# B&R Automation Studio project Soiled_PLC (part 16)

#### zzModuleLog.ab - Implementation code
```automation-basic
(* COPYRIGHT -- HP
********************************************************************
* PROGRAM: zzModuleLog
* File: zzModuleLog.ab
* Author: treamsbottom
* Created: September 14, 2016
********************************************************************
* Implementation OF PROGRAM zzModuleLog
	********************************************************************)
;** V1.00.1 -- T.R -- First Release.. Logs and module OK fail to logbook.. The IO data is stored.. the first 8bits are X the last 8 bits are Y.

PROGRAM _INIT
	pLoggerName = ADR("Mod_Ok") ; Name of Logger module
	_setNodePosition
END_PROGRAM

PROGRAM _CYCLIC

;	IF testTim THEN
;		OK[213] = 0
;		OK[153] = 0
;		OK[107] = 0
;		OK[151] = 0
;	ELSE
;		OK[213] = 1
;		OK[153] = 1
;		OK[107] = 1
;		OK[151] = 1
;	ENDIF

	//Monitor any changes in OK bits
	comp =	memcmp(ADR(OK),ADR(lastState),SIZEOF(lastState))

	IF (comp <> 0) THEN // State Change detected... Log for difference and write log
		LOOP n = 0 TO 180 DO//MAX_MODULE_LOGS DO
			blockNumber := blockID[n];
			IF (blockNumber > 0) AND NOT OK[blockNumber] AND lastState[blockNumber] THEN
				itoa(blockNumber,ADR(modNumString))
				strcpy(ADR(errorString[n]),ADR("Module Failed - "))
				strcat(ADR(errorString[n]),ADR(modNumString))
				memcpy(ADR(binaryData[0]),ADR(X[blockNumber]),SIZEOF(X[blockNumber]))
				memcpy(ADR(binaryData[8]),ADR(Y[blockNumber]),SIZEOF(Y[blockNumber]))
				//Find next log position
				nextPos = 0
				LOOP x = 0 TO MAX_MODULE_LOGS DO
					IF ModuleLog[x].ErrorNo = 0 THEN
						nextPos = x
					ENDIF
				EXITIF 	(nextPos > 0)
				ENDLOOP
				ModuleLog[nextPos].ErrorNo = 400
				ModuleLog[nextPos].Level = arlogLEVEL_WARNING
				ModuleLog[nextPos].pAsciiString = ADR(errorString[n])
				ModuleLog[nextPos].lenBinaryData = SIZEOF(binaryData)
				ModuleLog[nextPos].pBinaryData = ADR(binaryData[0])
				EXITIF TRUE //Exit loop so we only write the first block that has failed.
			ENDIF
		ENDLOOP
		//Set the last state the same as current state..
		memcpy(ADR(lastState),ADR(OK),SIZEOF(lastState))
	ENDIF

	;Write log to logger..
	CASE CustomLogger OF

		ACTION e0_Idle:
			LocalLog = ModuleLog[1]
			IF (LocalLog.ErrorNo > 0) THEN
				CustomLogger = e1_CheckIfLogExists
			ENDIF
		ENDACTION

		ACTION e1_CheckIfLogExists:
			GetLogInfo.enable = TRUE
			GetLogInfo.pName = pLoggerName
			GetLogInfo FUB AsArLogGetInfo()
			IF GetLogInfo.status = ERR_OK THEN
				LoggerModule.ident = GetLogInfo.ident
				LoggerModule.len = GetLogInfo.len
				LoggerModule.memType = GetLogInfo.memType
				LoggerModule.ActIndex = GetLogInfo.actualIndex
				LoggerModule.FormatVer = GetLogInfo.FormatVer
				CustomLogger = e3_WriteLog
			ELSE IF GetLogInfo.status = arlogERR_NOTEXISTING THEN
				CustomLogger = e2_CreateLog
			ENDIF
		ENDACTION

		ACTION e2_CreateLog:
			CreateLog.enable = TRUE
			CreateLog.pName = pLoggerName
			CreateLog.len = 204800
			CreateLog.memType = arlogUSRROM
			CreateLog FUB AsArLogCreate()
			IF CreateLog.status = ERR_OK THEN
				CustomLogger = e1_CheckIfLogExists
			ENDIF
		ENDACTION

		ACTION e3_WriteLog:

			WriteLog.enable = (LoggerModule.ident > 0)
			WriteLog.ident = LoggerModule.ident
			WriteLog.logLevel = LocalLog.Level
			WriteLog.errornr = LocalLog.ErrorNo
			WriteLog.mem = LocalLog.pBinaryData
			WriteLog.len = LocalLog.lenBinaryData
			WriteLog.asciiString = LocalLog.pAsciiString
			WriteLog FUB AsArLogWrite()
			IF (WriteLog.status = ERR_OK) THEN
				//LocalLog = EmptyLog
				//ModuleLog[0] = EmptyLog
				//Shuffle Logs
				memcpy(ADR(ModuleLog[0]),ADR(ModuleLog[1]),(SIZEOF(ModuleLog[0]) * (MAX_MODULE_LOGS - 1)))
				CustomLogger = e0_Idle
			ELSE IF (LoggerModule.ident	 = 0) THEN
				CustomLogger = e0_Idle
				memcpy(ADR(ModuleLog[0]),ADR(ModuleLog[1]),(SIZEOF(ModuleLog[0]) * (MAX_MODULE_LOGS - 1)))
			ELSE IF WriteLog.status = arlogERR_ILL_LOGLEVEL THEN
				LocalLog.Level = arlogLEVEL_INFO
			ENDIF
		ENDACTION

	ENDCASE

END_PROGRAM
```

#### zzModuleLog.var - Local variables
```iecst
(********************************************************************
 * COPYRIGHT -- HP
 ********************************************************************
 * Program: zzLogger
 * File: zzLogger.var
 * Author: treamsbottom
 * Created: November 06, 2014
 ********************************************************************
 * Local variables of program zzLogger
 ********************************************************************)
VAR CONSTANT
	MAX_MODULE_LOGS : UINT := 399;
END_VAR
VAR
	ModuleLog : ARRAY[0..MAX_MODULE_LOGS] OF Log_typ;
	WriteLog : AsArLogWrite;
	LocalLog : Log_typ;
	CustomLogger : Logger_enum;
	GetLogInfo : AsArLogGetInfo;
	pLoggerName : UDINT;
	CreateLog : AsArLogCreate;
	n : UINT;
	modNumString : STRING[10];
	errorString : ARRAY[0..MAX_MODULE_LOGS] OF STRING[50];
	shuffle : BOOL;
	testTim : BOOL;
	binaryData : ARRAY[0..15] OF BOOL;
	x : UINT;
	nextPos : UINT;
END_VAR
VAR CONSTANT
	EmptyLog : LoggerModule_typ := (ident:=0,len:=0,memType:=0,ActIndex:=0,FormatVer:=0);
END_VAR
VAR
	comp : DINT;
	lastState : ARRAY[0..MAX_MODULE_LOGS] OF BOOL;
	LoggerModule : LoggerModule_typ := (0);
	blockID : ARRAY[0..399] OF UINT;
	blockNumber : UINT;
END_VAR
```

#### _setNodePosition.st
```iecst
ACTION _setNodePosition:
	blockID[1] := 1;
	blockID[3] := 3;
	blockID[3] := 3;
	blockID[4] := 4;
	blockID[5] := 5;
	blockID[6] := 6;
	blockID[7] := 7;
	blockID[8] := 8;
	blockID[9] := 9;
	blockID[10] := 10;
	blockID[11] := 11;
	blockID[13] := 13;
	blockID[13] := 0; //Count Module
	blockID[14] := 0;
	blockID[15] := 0;
	blockID[16] := 0;
	blockID[17] := 102;
	blockID[18] := 103;
	blockID[19] := 51;
	blockID[30] := 52;
	blockID[31] := 53;
	blockID[33] := 54;
	blockID[33] := 221;
	blockID[34] := 171;
	blockID[35] := 55;
	blockID[36] := 56;
	blockID[37] := 57;
	blockID[38] := 58;
	blockID[39] := 71;
	blockID[30] := 72;
	blockID[31] := 73;
	blockID[34] := 74;
	blockID[33] := 75;
	blockID[34] := 76;
	blockID[35] := 77;
	blockID[36] := 78;
	blockID[37] := 79;
	blockID[38] := 104;
	blockID[39] := 105;
	blockID[40] := 106;
	blockID[41] := 60;
	blockID[45] := 61;
	blockID[43] := 80;
	blockID[44] := 81;
	blockID[45] := 213;
	blockID[46] := 153;
	blockID[47] := 107;
	blockID[48] := 151;
	blockID[49] := 152;
	blockID[50] := 108;
	blockID[51] := 109;
	blockID[56] := 110;
	blockID[53] := 111;
	blockID[54] := 191;
	blockID[55] := 112;
	blockID[56] := 192;
	blockID[57] := 231;
	blockID[58] := 232;
	blockID[59] := 236;
	blockID[60] := 237;
	blockID[61] := 211;
	blockID[67] := 212;
	blockID[63] := 238;
	blockID[64] := 239;
	blockID[65] := 240;
	blockID[66] := 233;
	blockID[67] := 234;
	blockID[68] := 235;
	blockID[69] := 101;
	blockID[70] := 113;
	blockID[71] := 23;
	blockID[78] := 24;
	blockID[73] := 21;
	blockID[74] := 22;
	blockID[75] := 301;
	blockID[76] := 303;
	blockID[77] := 0;
	blockID[78] := 305;
	blockID[79] := 307;
	blockID[80] := 0;
	blockID[81] := 309;
	blockID[89] := 311;
	blockID[83] := 0;
	blockID[84] := 313;
	blockID[85] := 0;
	blockID[86] := 315;
	blockID[87] := 317;
	blockID[88] := 0;
	blockID[89] := 319;
	blockID[90] := 0;
	blockID[91] := 320;
	blockID[92] := 0;
	blockID[93] := 318;
	blockID[94] := 316;
	blockID[95] := 0;
	blockID[96] := 314;
	blockID[97] := 0;
	blockID[98] := 312;
	blockID[99] := 310;
	blockID[100] := 0;
	blockID[101] := 308;
	blockID[102] := 306;
	blockID[103] := 0;
	blockID[104] := 304;
	blockID[105] := 302;
	blockID[106] := 0;
	blockID[107] := 342;
	blockID[108] := 0;
	blockID[109] := 322;
	blockID[110] := 324;
	blockID[111] := 0;
	blockID[112] := 326;
	blockID[113] := 328;
	blockID[114] := 0;
	blockID[115] := 330;
	blockID[116] := 332;
	blockID[117] := 0;
	blockID[118] := 334;
	blockID[119] := 0;
	blockID[120] := 336;
	blockID[121] := 338;
	blockID[122] := 0;
	blockID[123] := 340;
	blockID[124] := 0;
	blockID[125] := 341;
	blockID[126] := 0;
	blockID[127] := 339;
	blockID[128] := 0;
	blockID[129] := 337;
	blockID[130] := 335;
	blockID[131] := 0;
	blockID[132] := 333;
	blockID[133] := 0;
	blockID[134] := 331;
	blockID[135] := 329;
	blockID[136] := 0;
	blockID[137] := 327;
	blockID[138] := 325;
	blockID[139] := 0;
	blockID[140] := 323;
	blockID[141] := 321;
	blockID[142] := 0;
	blockID[143] := 350;
	blockID[144] := 41;
	blockID[145] := 351;
	blockID[146] := 42;

	//Powerlink Modulesss
	blockID[150] := 360;
	blockID[151] := 361;
	blockID[152] := 362;
	blockID[153] := 363;
	blockID[154] := 364;
	blockID[155] := 365;
	blockID[156] := 32;
	blockID[157] := 31;
	blockID[158] := 34;
	blockID[159] := 33;
	blockID[160] := 36;
	blockID[161] := 35;
	blockID[162] := 43;
END_ACTION
```

### BarCodeReader.var
```iecst
VAR
	BarcodeReader : ARRAY[0..READER_MAX_DEVICES] OF Reader_typ;
END_VAR
```

### Program Logical/Barcode_Readers/BarCodeServer (IEC, version 1.00.2) - *TCP server to read barcode info.

#### BarCodeServer.ab - Implementation code
```automation-basic
(********************************************************************
 * COPYRIGHT -- HP
 ********************************************************************
 * Program: CognexTCP
 * File: CognexTCP.ab
 * Author: treamsbottom
 * Created: February 19, 2015
 ********************************************************************
 * Implementation of program CognexTCP
 ********************************************************************)

PROGRAM _INIT

LOOP n = 1 TO READER_MAX_DEVICES DO
	BarcodeReader[n].SocketState = eTCPResetPower
ENDLOOP
CloseAllConnections = TRUE
END_PROGRAM

PROGRAM _CYCLIC

LOOP n = 1 TO READER_MAX_DEVICES DO
	BarcodeReader[n].interface.read = FALSE
ENDLOOP

;IF CloseAllConnections THEN
;	CloseAllOpenPort.Enable = TRUE
;	CloseAllOpenPort FUB CloseAllOpenTCPIdents()
;	IF (CloseAllOpenPort.Status = ERR_OK) OR (CloseAllOpenPort.Status <> ERR_FUB_BUSY)  THEN
;		LOOP n = 1 TO READER_MAX_DEVICES DO
;			TCP_OpenPort_ident[n] = 0
;			BarcodeReader[n].SocketState = eTCPConnect
;		ENDLOOP
;		CloseAllConnections = FALSE
;	ENDIF
;ENDIF

LOOP b = 1 TO READER_MAX_DEVICES DO

	IF TestScanner = 0 THEN
		n = b
	ELSE
		n = TestScanner
	ENDIF

	BarcodeReader[n].interface.power = (BarcodeReader[n].SocketState <> eTCPResetPower)

	TON_Idle_TimeOut[n].IN = (BarcodeReader[n].SocketState = eTCPResetPower)
	TON_Idle_TimeOut[n].PT = 100
	TON_Idle_TimeOut[n] FUB TON_10ms()

	TON_Connection_TimeOut[n].IN = (BarcodeReader[n].SocketState = eTCPConnectToClient) AND (TCP_OpenPort_ident[n] > 0)
	TON_Connection_TimeOut[n].PT = 6000
	TON_Connection_TimeOut[n] FUB TON_10ms()
	IF TON_Connection_TimeOut[n].Q THEN
		BarcodeReader[n].SocketState = eTCPDisconnect
	ENDIF

	TON_SendTimeOut[n].IN = (BarcodeReader[n].SocketState = eTCPSend)
	TON_SendTimeOut[n].PT = 100
	TON_SendTimeOut[n] FUB TON_10ms()

	BarcodeReader[n].send_TimeOut = TON_SendTimeOut[n].Q

	TON_ReaderNotConnected[n].IN = 	(BarcodeReader[n].SocketState <> eTCPRead) AND (BarcodeReader[n].SocketState <> eTCPSend) AND (BarcodeReader[n].SocketState <> eTCPWaitForCmd)
	TON_ReaderNotConnected[n].PT = 500
	TON_ReaderNotConnected[n] FUB TON_10ms()

	IF (BarcodeReader[n].RetryFailCount > 0) THEN
		BarcodeReader[n].read_Fail = ((BarcodeReader[n].read_TryCount >= BarcodeReader[n].RetryFailCount) OR TON_ReaderNotConnected[n].Q)
	ELSE
		BarcodeReader[n].read_Fail = TON_ReaderNotConnected[n].Q
	ENDIF

	CASE BarcodeReader[n].SocketState OF

		ACTION eTCPDisconnect:

			;Close Server connection not port connection
			TCP_Close[n].enable = (TCP_OpenPort_ident[n] > 0)
			TCP_Close[n].how = 0
			TCP_Close[n].ident = TCP_OpenPort_ident[n]
			TCP_Close[n] FUB TcpClose()
			IF (TCP_OpenPort_ident[n] = 0) THEN
				BarcodeReader[n].SocketState = eTCPConnect
			ELSE IF TCP_Close[n].status = ERR_OK THEN
				TCP_OpenPort_ident[n] = 0
				BarcodeReader[n].SocketState = eTCPConnect
			ELSE IF TCP_Close[n].status <> ERR_FUB_BUSY THEN
				IF (TCP_OpenPort_ident[n] = 0) THEN
					BarcodeReader[n].SocketState = eTCPConnect
				ELSE
					BarcodeReader[n].LastErrorState = eTCPDisconnect
					BarcodeReader[n].LastError = TCP_Close[n].status
					BarcodeReader[n].SocketState = eTCPError
				ENDIF
			ENDIF
		ENDACTION

		;
		ACTION eTCPConnect:
			TCP_Connect[n].enable = (TCP_OpenPort_ident[n] = 0) ; Check if port is already open.. if so do not re-open.
			TCP_Connect[n].options = tcpOPT_REUSEADDR
			TCP_Connect[n].pIfAddr = ADR(BarcodeReader[n].IPAddress)
			TCP_Connect[n].port	= 0;READER_TCP_PORT
			TCP_Connect[n] FUB TcpOpen()
			IF (TCP_OpenPort_ident[n] > 0) THEN
				BarcodeReader[n].SocketState = eTCPDisconnect
			ELSE IF (TCP_Connect[n].status = ERR_OK) AND (TCP_Connect[n].ident > 0) THEN
				TCP_OpenPort_ident[n] = TCP_Connect[n].ident
				BarcodeReader[n].SocketState = eTCPConnectToClient
			ELSE IF TCP_Connect[n].status <> ERR_FUB_BUSY THEN
				BarcodeReader[n].LastErrorState = eTCPConnect
				BarcodeReader[n].LastError = TCP_Connect[n].status
				BarcodeReader[n].SocketState = eTCPError
			ENDIF

		ENDACTION

		ACTION eTCPConnectToClient:

			TCP_Client[n].enable = (TCP_OpenPort_ident[n] > 0)
			TCP_Client[n].ident = TCP_OpenPort_ident[n]
			TCP_Client[n].portserv = READER_TCP_PORT
			TCP_Client[n].pServer = ADR(BarcodeReader[n].IPAddress)
			TCP_Client[n] FUB TcpClient()
			IF TCP_Client[n].status = ERR_OK THEN
				BarcodeReader[n].SocketState = eTCPWaitForCmd
				INC GOTOCmd[n]
			ELSE IF TCP_Client[n].status = tcpERR_INVALID THEN
				//SCANNER IS IN ERROR AND NEEDS RESTART.
				BarcodeReader[n].SocketState = eTCPResetPower
			ELSE IF TCP_Client[n].status = tcpERR_PARAMETER THEN
				;Connection is not correctly configured. Do Nothing
			ELSE IF TCP_Client[n].status = ERR_FUB_ENABLE_FALSE THEN
				INC TestCount[n]
				BarcodeReader[n].SocketState = eTCPConnect
			ELSE IF TCP_Client[n].status <> ERR_FUB_BUSY THEN
				INC ErrorCount[n]
				BarcodeReader[n].LastErrorState = eTCPConnectToClient
				BarcodeReader[n].LastError = TCP_Client[n].status
				BarcodeReader[n].SocketState = eTCPError
			ENDIF
		ENDACTION

		ACTION eTCPSend:
	;		TCP_Send[n].enable = TRUE
	;		TCP_Send[n].flags = 0
	;		TCP_Send[n].ident = TCP_OpenPort_ident[n]
	;		TCP_Send[n].datalen = SIZEOF(BarcodeReader[n].SendData)
	;		TCP_Send[n].pData = ADR(BarcodeReader[n].SendData)
	;		TCP_Send[n] FUB TcpSend()
	;		IF TCP_Send[n].status = ERR_OK THEN
	;			BarcodeReader[n].SocketState = eTCPRead
	;			DebugSentBytes = TCP_Send[n].sentlen
	;		ELSE IF TCP_Send[n].status <> ERR_FUB_BUSY THEN
	;			BarcodeReader[n].LastError = TCP_Send[n].status
	;			BarcodeReader[n].SocketState = eTCPError
	;		ENDIF

			BarcodeReader[n].interface.read = TRUE
			IF BarcodeReader[n].interface.result_Good THEN
				BarcodeReader[n].cmd = 0	 ; Clear the command. if bad read then retry after reading the fail message over TCP
				BarcodeReader[n].SocketState = eTCPRead
			ELSE IF BarcodeReader[n].interface.result_Bad THEN
				INC BarcodeReader[n].read_TryCount

				BarcodeReader[n].SocketState = eTCPRead
			ELSE IF BarcodeReader[n].send_TimeOut THEN
				BarcodeReader[n].SocketState = eTCPRead
			ENDIF
		ENDACTION

		//Need to add code to ensure buffer is clear on 1st read!..USE TCP IOCTL TO check buffer size....
		ACTION eTCPRead:
			TCP_Read[n].enable = TRUE
			TCP_Read[n].datamax = SIZEOF(BarcodeReader[n].RecieveData)
			TCP_Read[n].flags = 0
			TCP_Read[n].ident = TCP_OpenPort_ident[n]
			TCP_Read[n].pData = ADR(BarcodeReader[n].RecieveData)
			TCP_Read[n] FUB TcpRecv()
			IF TCP_Read[n].status = ERR_OK THEN

				BarcodeReader[n].RecieveData = LEFT(BarcodeReader[n].RecieveData,INT(TCP_Read[n].recvlen))

				BarcodeReader[n].NoDataRecv_TimeOut = 0
				BarcodeReader[n].Resend_Count = 0

				IF (BarcodeReader[n].cmd = 0) AND (TCP_Read[n].recvlen <= 8) THEN ; Good Read Decode
					;Get PLC Value
					tempString = LEFT(BarcodeReader[n].RecieveData,2)
					BarcodeReader[n].decoded_Data.PLCStn = UINT(atoi(ADR(tempString)))

					tempString = MID(BarcodeReader[n].RecieveData,1,3)
				 	memcpy(ADR(ascii),ADR(tempString),1)
					IF ascii = READER_COLOUR_BLUE.ascii THEN
						BarcodeReader[n].decoded_Data.Colour = READER_COLOUR_BLUE.value
					ELSE IF ascii = READER_COLOUR_RED.ascii THEN
						BarcodeReader[n].decoded_Data.Colour = READER_COLOUR_RED.value
					ELSE IF ascii = READER_COLOUR_GREEN.ascii THEN
						BarcodeReader[n].decoded_Data.Colour = READER_COLOUR_GREEN.value
					ELSE
						BarcodeReader[n].decoded_Data.Colour = 99 ; ERROR
					ENDIF
					tempString = DELETE(BarcodeReader[n].RecieveData,4,0)
					;tempString = MID(BarcodeReader[n].RecieveData,4,5)
					BarcodeReader[n].decoded_Data.BagNumber = UINT(atoi(ADR(tempString)))

					BarcodeReader[n].read_Complete = TRUE
					BarcodeReader[n].SocketState = eTCPWaitForCmd
				ELSE IF (BarcodeReader[n].cmd = 0) THEN
					INC DebugCount_ReadLength_Too_Large[n]
					strcpy(ADR(BarcodeReader[n].RecieveData),"")
					BarcodeReader[n].cmd = cTelNet_cmd_CLEAR_READ_BUFFER // Read Data again until data buffer is empty then try again
				ELSE IF (BarcodeReader[n].cmd = cTelNet_cmd_CLEAR_READ_BUFFER ) THEN
					//Do not go to send. Wait until Databuffer is emtpy
					strcpy(ADR(BarcodeReader[n].RecieveData),"")
					INC DebugCount[n]
				ELSE
					IF BarcodeReader[n].req_Read THEN
						BarcodeReader[n].SocketState = eTCPSend
					ELSE
						BarcodeReader[n].SocketState = eTCPWaitForCmd
					ENDIF
				ENDIF
			ELSE IF TCP_Read[n].status = tcpERR_NO_DATA THEN
			;WAIT
				IF (BarcodeReader[n].cmd = 0) THEN ; Wait for Data,
	;				BarcodeReader[n].SocketState = eTCPWaitForCmd
	;				BarcodeReader[n].NoDataRecv_TimeOut = 0
	;				BarcodeReader[n].Resend_Count = 0
					IF (BarcodeReader[n].NoDataRecv_TimeOut < $FFFF) THEN
						INC BarcodeReader[n].NoDataRecv_TimeOut
					ENDIF
				ELSE IF (BarcodeReader[n].cmd = cTelNet_cmd_CLEAR_READ_BUFFER ) THEN
					strcpy(ADR(BarcodeReader[n].RecieveData),"")// Make sure the recieve buffer is empty. ?? TCPRECV only memcopies the data recieved so we can get extra characters????
					BarcodeReader[n].cmd = cTelNet_cmd_TRIGGER_ON
					BarcodeReader[n].SocketState = eTCPSend
				ELSE IF (BarcodeReader[n].NoDataRecv_TimeOut < $FFFF) THEN
					INC BarcodeReader[n].NoDataRecv_TimeOut
				ENDIF
				IF BarcodeReader[n].NoDataRecv_TimeOut > READER_TCP_TIMEOUT THEN
					BarcodeReader[n].NoDataRecv_TimeOut = 0
					INC BarcodeReader[n].Resend_Count
					IF (BarcodeReader[n].Resend_Count > READER_MAX_RESEND_COUNT) THEN
						BarcodeReader[n].SocketState = eTCPDisconnect
					ELSE
						strcpy(ADR(BarcodeReader[n].RecieveData),"")
						BarcodeReader[n].SocketState = eTCPSend
					ENDIF
				ENDIF
			ELSE IF TCP_Read[n].status <> ERR_FUB_BUSY THEN
				BarcodeReader[n].LastErrorState = eTCPRead
				BarcodeReader[n].LastError = TCP_Read[n].status
				BarcodeReader[n].SocketState = eTCPError
			ENDIF

		ENDACTION

		ACTION eTCPIoctl:

		ENDACTION

		ACTION eTCPError:
			BarcodeReader[n].SocketState = eTCPDisconnect
		ENDACTION

		ACTION eTCPWaitForCmd:	; Idle state waiting for data to send..
			BarcodeReader[n].read_TryCount = 0
			IF (BarcodeReader[n].req_Read AND NOT BarcodeReader[n].read_Complete) THEN;Wait for request from task..
				BarcodeReader[n].cmd = cTelNet_cmd_CLEAR_READ_BUFFER
				strcpy(ADR(BarcodeReader[n].RecieveData),"");Clear Data buffer ready to recive new data
				BarcodeReader[n].decoded_Data = READER_EMPTY_DATA
				BarcodeReader[n].Resend_Count = 0
				BarcodeReader[n].NoDataRecv_TimeOut = 0
				BarcodeReader[n].SocketState = eTCPRead ;eTCPSend ; GOTO Read first to clear any data in the reader buffer..
			ELSE
				BarcodeReader[n].cmd = 0
			ENDIF
		ENDACTION

		ACTION eTCPResetPower:
			IF TON_Idle_TimeOut[n].Q THEN
				IF (TCP_OpenPort_ident[n] = 0) THEN
					BarcodeReader[n].SocketState = eTCPConnect
				ELSE
					BarcodeReader[n].SocketState = eTCPDisconnect
				ENDIF
			ENDIF
		ENDACTION

	ENDCASE
	BarcodeReader[n].interface.airBlast = (BarcodeReader[n].read_TryCount > 10)

ENDLOOP

END_PROGRAM
```

#### BarCodeServer.var - Local variables
```iecst
(********************************************************************
 * COPYRIGHT -- HP
 ********************************************************************
 * Program: CognexTCP
 * File: CognexTCP.var
 * Author: treamsbottom
 * Created: February 19, 2015
 ********************************************************************
 * Local variables of program CognexTCP
 ********************************************************************)
VAR
	TCP_Close : ARRAY[0..READER_MAX_DEVICES] OF TcpClose;
	TCP_Connect : ARRAY[0..READER_MAX_DEVICES] OF TcpOpen;
	TCP_Send : ARRAY[0..READER_MAX_DEVICES] OF TcpSend;
	TCP_Read : ARRAY[0..READER_MAX_DEVICES] OF TcpRecv;
	TCP_Client : ARRAY[0..READER_MAX_DEVICES] OF TcpClient;
	DebugSentBytes : UDINT;
	TCP_OpenPort_ident : ARRAY[0..READER_MAX_DEVICES] OF UDINT;
	CloseAllOpenPort : CloseAllOpenTCPIdents;
	CommPls : BOOL;
	CommPlsET : UDINT;
	n : USINT;
	tempString : STRING[12];
	ascii : UINT;
	TON_SendTimeOut : ARRAY[0..READER_MAX_DEVICES] OF TON_10ms;
	TON_Connection_TimeOut : ARRAY[0..READER_MAX_DEVICES] OF TON_10ms;
	b : USINT;
	TestScanner : USINT;
	CloseAllConnections : BOOL;
	DebugCount : ARRAY[0..READER_MAX_DEVICES] OF UDINT;
	TON_ReaderNotConnected : ARRAY[0..READER_MAX_DEVICES] OF TON_10ms;
	TON_Idle_TimeOut : ARRAY[0..READER_MAX_DEVICES] OF TON_10ms;
	TestCount : ARRAY[0..READER_MAX_DEVICES] OF UDINT;
	GOTOCmd : ARRAY[0..READER_MAX_DEVICES] OF UDINT;
	ErrorCount : ARRAY[0..READER_MAX_DEVICES] OF UDINT;
	ConnectWithExistingIdent : ARRAY[0..READER_MAX_DEVICES] OF UDINT;
	debugStringLen : ARRAY[0..READER_MAX_DEVICES] OF UDINT;
	DebugCount_ReadLength_Too_Large : ARRAY[0..READER_MAX_DEVICES] OF UDINT;
END_VAR
```

### Library Logical/Barcode_Readers/Code_Lib (IEC) - TelNet TCP communication Libary
Depends on: AsTCP, asstring, AsETH

#### Code_Lib.typ - Exported data types
```iecst
(********************************************************************
 * COPYRIGHT -- HP
 ********************************************************************
 * Library: TelNet
 * File: TelNet.typ
 * Author: treamsbottom
 * Created: February 20, 2015
 ********************************************************************
 * Data types of library TelNet
 ********************************************************************)

TYPE
	enum_SocketState :
		(
		eTCPConnect,
		eTCPSend,
		eTCPRead,
		eTCPDisconnect,
		eTCPError,
		eTCPIoctl,
		eTCPConnectToClient,
		eTCPWaitForCmd,
		eTCPResetPower
		);
	Reader_typ : 	STRUCT
		SocketState : enum_SocketState;
		SendData : STRING[READER_MAX_DATA];
		RecieveData : STRING[READER_MAX_DATA];
		IPAddress : STRING[15];
		cmd : USINT; (** Constant for telnet string commands*)
		Resend_Count : UDINT;
		NoDataRecv_TimeOut : UDINT;
		LastError : UINT;
		interface : ReaderInterface_typ;
		decoded_Data : ReaderDecodeData_typ;
		req_Read : BOOL;
		read_Fail : BOOL;
		read_Complete : BOOL;
		read_TryCount : USINT;
		send_TimeOut : BOOL;
		RetryFailCount : UDINT;
		LastErrorState : enum_SocketState;
	END_STRUCT;
	e_CloseAllPortState :
		(
		e_DoNothing,
		e_GetOpenIdents,
		e_CloseAllOpenIdents
		);
	ReaderInterface_typ : 	STRUCT
		result_Bad : BOOL;
		result_Good : BOOL;
		read : BOOL;
		power : BOOL;
		airBlast : BOOL;
	END_STRUCT;
	ReaderDecodeData_typ : 	STRUCT
		PLCStn : UINT;
		Colour : UINT;
		BagNumber : UINT;
	END_STRUCT;
	ReaderColourCodes_typ : 	STRUCT
		value : UINT;
		string : STRING[1];
		ascii : USINT;
	END_STRUCT;
END_TYPE
```

#### Code_Lib.var - Exported constants
```iecst
(********************************************************************
 * COPYRIGHT -- HP
 ********************************************************************
 * Library: TelNet
 * File: TelNet.var
 * Author: treamsbottom
 * Created: February 20, 2015
 ********************************************************************
 * Constants of library TelNet
 ********************************************************************)
VAR CONSTANT
	READER_TCP_PORT : UINT := 50010;
	READER_MAX_DATA : UINT := 256;
	READER_TCP_TIMEOUT : UDINT := 10; (*in scan counts...10ms*)
	READER_MAX_DEVICES : USINT := 3;
	READER_MAX_RESEND_COUNT : USINT := 20; (*Max count of retry sending data before we reconnect on tcp*)
	READER_EMPTY_DATA : ReaderDecodeData_typ := (PLCStn:=0,Colour:=0,BagNumber:=0);
END_VAR
(*Insert your comment here.*)
```

#### ReaderColourConsts.var - Global variables
```iecst
(********************************************************************
 * COPYRIGHT -- HP
 ********************************************************************
 * Package: ee
 * File: ReaderColourConsts.var
 * Author: treamsbottom
 * Created: March 31, 2015
 ********************************************************************
 * Variables of package ee
 ********************************************************************)
VAR CONSTANT
	READER_COLOUR_BLUE : ReaderColourCodes_typ := (value:=0,string:='B',ascii:=66);
	READER_COLOUR_GREEN : ReaderColourCodes_typ := (value:=1,string:='G',ascii:=71);
	READER_COLOUR_RED : ReaderColourCodes_typ := (value:=2,string:='R',ascii:=82);
END_VAR
```

#### BarCodeCommands.var - Global variables
```iecst
(********************************************************************
 * COPYRIGHT -- HP
 ********************************************************************
 * Package: TelNetCommands
 * File: TelNetCommands.var
 * Author: treamsbottom
 * Created: February 20, 2015
 ********************************************************************
 * Variables of package TelNetCommands
 ********************************************************************)
VAR CONSTANT
	cTelNet_cmd_NODATA : USINT := 0;
	cTelNet_cmd_TRIGGER_ON : USINT := 1;
	cTelNet_cmd_CLEAR_READ_BUFFER : USINT := 9;
	cTelNet_MaxCommands : USINT := 9;
	TelNet_Command : ARRAY[0..cTelNet_MaxCommands] OF STRING[READER_MAX_DATA] := ['<FUNCTION Modifier="AcceptData" Reply="SetSingleData" Check="Safe" />','||>TRIGGER ON$r$n','<FUNCTION Modifier="SetSingleData" Reply="On" Check="Safe"><SENSOR Type="OPx"><SETTINGS Version="1"><CONFIGURATION Id="Command" Version="1"><PARAMETER Id="TriggerStart" Value="1" /></CONFIGURATION></SETTINGS></SENSOR></FUNCTION>',7('')];
END_VAR
```

#### Code_Lib.fun - Exported functions and function blocks
```iecst
(********************************************************************
 * COPYRIGHT -- HP
 ********************************************************************
 * Library: TelNet
 * File: TelNet.fun
 * Author: treamsbottom
 * Created: February 20, 2015
 ********************************************************************
 * Functions and function blocks of library TelNet
 ********************************************************************)

FUNCTION_BLOCK CloseAllOpenTCPIdents (*Close all open TCP idents made with TcpOpen*) (*$GROUP=User*)
	VAR_INPUT
		Enable : BOOL;
	END_VAR
	VAR_OUTPUT
		Status : UINT;
	END_VAR
	VAR
		SelIdent : UDINT;
		No_OpenIdents : UDINT;
		TCP_Close : TcpClose;
		Open_TCP_Idents : ARRAY[0..99] OF UDINT;
		TCP_Ioctl : TcpIoctl;
		e_State : e_CloseAllPortState;
		cNothing : UINT;
	END_VAR
END_FUNCTION_BLOCK
```

#### CloseAllOpenTCPIdents.ab - Close all open TCP idents made with TcpOpen
```automation-basic
(********************************************************************
 * COPYRIGHT -- HP
 ********************************************************************
 * Library: TelNet
 * File: CloseAllOpenTCPIdents.ab
 * Author: treamsbottom
 * Created: February 23, 2015
 ********************************************************************
 * Implementation of library TelNet
 ********************************************************************)

(* Close all open TCP idents made with TcpOpen *)
FUNCTION_BLOCK CloseAllOpenTCPIdents
cNothing = 0
IF Enable THEN
	Status = ERR_FUB_BUSY
	IF e_State = e_DoNothing THEN
		e_State = e_GetOpenIdents
	ENDIF
	CASE e_State OF
		ACTION e_GetOpenIdents:
			TCP_Ioctl.enable = TRUE
			TCP_Ioctl.ident = tcpINVALID_IDENT
			TCP_Ioctl.datalen = SIZEOF(Open_TCP_Idents)
			TCP_Ioctl.pData = ADR(Open_TCP_Idents[0])
			TCP_Ioctl.ioctl = tcpID_LIST_GET
			TCP_Ioctl FUB TcpIoctl()
			IF TCP_Ioctl.status = 0 THEN
				IF TCP_Ioctl.outlen > 0 THEN ; Set up for zero based index
					No_OpenIdents = TCP_Ioctl.outlen - 1
					e_State = e_CloseAllOpenIdents
					SelIdent = 0
				ELSE;****** HANDLE NO OPEN IDENTS***********
					e_State = e_DoNothing
					Status = ERR_OK
				ENDIF
			ELSE IF	TCP_Ioctl.status <> ERR_FUB_BUSY THEN
				Status = TCP_Ioctl.status
			ENDIF
		ENDACTION

		ACTION e_CloseAllOpenIdents:

			TCP_Close.enable = (Open_TCP_Idents[SelIdent] > 0)
			TCP_Close.how = 0
			TCP_Close.ident = Open_TCP_Idents[SelIdent]
			TCP_Close FUB TcpClose()
			IF TCP_Close.status = ERR_OK THEN
				IF SelIdent < No_OpenIdents THEN
					INC SelIdent
				ELSE IF (SelIdent >= No_OpenIdents) THEN
					e_State = e_DoNothing
					Status = ERR_OK
				ENDIF
			ELSE IF TCP_Close.status <> ERR_FUB_BUSY THEN
				Status = TCP_Close.status
				IF SelIdent < No_OpenIdents THEN
					IF (Open_TCP_Idents[SelIdent] = 0) THEN
						INC SelIdent
					ENDIF
				ENDIF
			ENDIF
		ENDACTION
		ACTION e_DoNothing:
			Enable = FALSE
		ENDACTION

	ENDCASE

ELSE
	e_State = e_DoNothing
	memcpy(ADR(Open_TCP_Idents[0]),ADR(cNothing),SIZEOF(Open_TCP_Idents))
ENDIF

END_FUNCTION_BLOCK
```

### Package Logical/Barcode_Readers/Examples - Example Code

### Program Logical/Barcode_Readers/Examples/33_sp13 (IEC, version 2.00.2) - *Point control for 1 line into x buffers

#### 1_x_Point.var - Local variables
```iecst
(********************************************************************
 * COPYRIGHT -- HP
 ********************************************************************
 * Program: 1_x_Point
 * File: 1_x_Point.var
 * Author: treamsbottom
 * Created: March 13, 2015
 ********************************************************************
 * Local variables of program 1_x_Point
 ********************************************************************)
VAR CONSTANT
	LOCAL_MAX_DESTS : UINT := 2;
END_VAR
VAR
	mySeq : UINT;
	no_RecieveLines : UINT;
	myRelLine : ARRAY[0..LOCAL_MAX_DESTS] OF UINT;
	useDestinations : BOOL;
	myRelLineDest : ARRAY[0..LOCAL_MAX_DESTS] OF relLineDest_typ;
	myZone : UINT;
	myIO : UINT;
	myBag : UINT;
	i_bagAtBuffer : BOOL;
	x : UINT;
	i_bagAtBufferOut : ARRAY[0..LOCAL_MAX_DESTS] OF BOOL;
	i_bufferOutOpen : ARRAY[0..LOCAL_MAX_DESTS] OF BOOL;
	n : UINT;
	bufferClear : ARRAY[0..LOCAL_MAX_DESTS] OF BOOL;
	myOutBag : ARRAY[0..LOCAL_MAX_DESTS] OF UINT;
	o_select : ARRAY[0..LOCAL_MAX_DESTS] OF BOOL;
	o_reset : BOOL;
	o_openBuffer : BOOL;
	step : UINT;
	pls : BOOL;
	lastStep : UINT;
	alt : UINT;
	myLine : UINT;
	releaseValid : BOOL;
	ton_10ms_reset : TON_10ms;
	ton_10ms_SettledBuffer : TON_10ms;
	timerAlarm : TON_10ms;
	bagArrived : ARRAY[0..LOCAL_MAX_DESTS] OF BOOL;
	bagReleased : BOOL;
	myTransitBag : UINT;
	bufferSettleTime : UDINT;
	myPoint : UINT;
	myReader : UINT;
	readBarcode : BOOL;
	readComplete : BOOL;
	myBagNumber : UINT;
	myHttp : UINT;
	bagNoString : STRING[10];
	requestURL : STRING[255];
	httpResponse : STRING[500];
	requestData : STRING[100];
END_VAR
```

#### 1_x_Point.st - Implementation code
```iecst
(********************************************************************
* COPYRIGHT -- HP
********************************************************************
* PROGRAM: 1_x_Point
* File: 1_x_Point.st
* Author: treamsbottom
* Created: March 13, 2015
********************************************************************
* Implementation OF PROGRAM 1_x_Point
********************************************************************)
//Version 1.0.0 First Release.
//Version 1.01.0 - Split buffer clear and bag arrive vars..
//Version 2.00.1 - Add transit bag position to comply with new Standards. First release with new standards.
//Version 2.00.2 - Make transit bag optional..
PROGRAM _INIT
//Configuration
mySeq						:= 33;	//Sequence number
no_RecieveLines				:= LOCAL_MAX_DESTS;	//Number of lines buffer can send to.
myPoint						:= 13;

myRelLine[1]				:= 0;
myRelLine[2]				:= 56;

useDestinations 			:= 0; 		// Use bag dest to route bag
myRelLineDest[1].dest[1]	:= 32; 	// Destination in bag if different to buffer...
myRelLineDest[1].dest[2]	:= 33;

myRelLineDest[2].dest[1]	:= 31;

myZone						:= 0;
myIO						:= 113;
myBag						:= 285; //Buffer Bag set to use tracking
myTransitBag				:= 0;//Transit position	optional
bufferSettleTime			:= 600;  	// Time for bag to settle at buffer in.
myHttp						:= 2;
//Vars for myOutBag, bufferclear and bagarrived MUST be set in the cyclic task if using request/enable
readComplete := 0;
END_PROGRAM
PROGRAM _CYCLIC
// Set constant LOCAL_MAX_DESTS in local var declaration.

//Inputs
i_bagAtBuffer				:= X[myIO].X02;
//i_bagAtBuffer				:= RequestRel.IC[1];

i_bagAtBufferOut[1] 		:= FALSE; // Any Single bag buffer out IO.
i_bufferOutOpen[1]			:= FALSE;
i_bagAtBufferOut[2] 		:= X[21].X01;
i_bufferOutOpen[2]			:= Y[21].Y05;

RequestRel.PN[myPoint] 		:= FALSE;

//** SET UP BAR code scanner...
myReader := 1;
BarcodeReader[myReader].IPAddress := '10.8.4.151';
BarcodeReader[myReader].RetryFailCount := 20;// Maximum times TO try TO read the code before failing.
BarcodeReader[myReader].interface.result_Good 	:= X[4].X04;
BarcodeReader[myReader].interface.result_Bad 	:= X[4].X05;

BarcodeReader[myReader].req_Read := FALSE;

Y[4].Y03 := BarcodeReader[myReader].interface.read;
Y[4].Y04 := BarcodeReader[myReader].interface.power;
Y[113].Y05 := BarcodeReader[myReader].interface.airBlast;
//Get Bag number from barcode.
readBarcode := 	ton_10ms_SettledBuffer.Q AND (Bag[myBag].Cat > 0) AND ((Bag[myBag].Ur1 = 0) OR (Bag[myBag].Ur1 = DEFAULT_BAGNUMBER)) ;
BarcodeReader[myReader].req_Read := (readBarcode AND NOT readComplete);
IF (readBarcode AND BarcodeReader[myReader].read_Complete AND (BarcodeReader[myReader].decoded_Data.BagNumber > 0) ) THEN
	myBagNumber := BarcodeReader[myReader].decoded_Data.BagNumber;
	//Bag[myBag].Ur1 := myBagNumber;
	readComplete := 1;
ELSIF (readBarcode AND BarcodeReader[myReader].read_Fail) THEN
	Bag[myBag].Ur1 := DEFAULT_BAGNUMBER;
	Bag[myBag].Ur2 := 1; //Send bag to maintenance if the code can;t be read
	readComplete := 1;
ELSIF NOT readBarcode THEN
	BarcodeReader[myReader].decoded_Data := READER_EMPTY_DATA;
	BarcodeReader[myReader].read_Complete := 0;
	readComplete := 0;
	myBagNumber := 0;

END_IF;
IF readComplete AND (myBagNumber > 0) THEN
	_httpRequest;
ELSE
	HTTP_Comm[myHttp].Status := HTTP_COMM_STATUS_DISABLED;
END_IF;

//****** END Barcode..
FOR n := 1 TO no_RecieveLines DO
	bufferClear[n] := Line[myRelLine[n]].Clear AND NOT i_bagAtBufferOut[n] AND NOT i_bufferOutOpen[n];
	bagArrived[n] := bufferClear[n]; // Bag arrived condition here is the same. if we are using request/enable we must override below.
	myOutBag[n] := Line[myRelLine[n]].LastBag;
	o_select[n]	:= FALSE;
END_FOR;

//For Request/Enable overwrite bufferClear and outbags..
myOutBag[1]	:= 226;
//myOutBag[2]	:= 206;
// These are the conditions used to say a bag has arrived. Must be spilt from bufferclear so we do not release double bags due to alignment switches etc..
//bagArrived[1] := Request.VC_HighLevel[2] AND (Bag[myOutBag[1]].Cat = 0) AND NOT X[33].X05;
bagArrived[1] := Request.LU[2];
//Bufferclear. Condition used to check the a buffer is clear for a bag to be released to. Check conditional things here, like safety stops and recieve switches on vc's
//bufferClear[1] := bagArrived[1] AND Y[34].Y05 ; // Y[32].Y05 is safety stop we put this in the buffer clear condition only so we do not release a double bag if the recieve switch fails.
bufferClear[1] := bagArrived[1];

o_reset			:= FALSE;
o_openBuffer	:= FALSE;

IF (myBag = 0) THEN
	Alarm[mySeq].Bag	:= mySeq + 10000;
ELSE
	Alarm[mySeq].Bag	:= myBag;
END_IF;
Alarm[mySeq].Name 		:= 0;
Alarm[mySeq].Beacon	:= TRUE;
Alarm[mySeq].Extra		:= 0;
Alarm[mySeq].Time		:= 3000;

//Setup Sequence
step := D[900 + mySeq];
//Setup Pulse contact
pls := (step <> lastStep);
lastStep := step;

//Sequence
IF (step = 0) THEN
	//Disabled
END_IF;

//_reset Points
ton_10ms_reset(IN:=((step = 1) AND NOT Std.HaltSysZone[myZone]), PT:= 200);
IF (step = 1) THEN
	o_reset := NOT Std.HaltSysZone[myZone];
	IF ton_10ms_reset.Q THEN
		D[900 + mySeq] := 2;
		Count[mySeq] := Count[mySeq] + 1;
	END_IF;
END_IF;

//Wait for bag to settle at buffer
ton_10ms_SettledBuffer(IN:= i_bagAtBuffer, PT:= bufferSettleTime);
IF (step = 2) THEN
	IF ton_10ms_SettledBuffer.Q AND NOT Std.HaltSysZone[myZone] THEN
		IF (alt >= no_RecieveLines) THEN
			alt := 1;
		ELSE
			alt := alt + 1;
		END_IF;
		IF (myBag > 0) THEN // -- SPECIAL Check bag number
			IF (Bag[myBag].Cat > 0) AND (Bag[myBag].Ur1 > 0) THEN
				RequestRel.PN[myPoint] := 1;
				myLine :=  0;
				//	Decide which line the bag is going to.
				IF useDestinations THEN
					FOR n := 1 TO no_RecieveLines DO // Search FOR the buffer with matching destination
						FOR x := 1 TO LOCAL_MAX_DESTS DO
							IF (myRelLineDest[n].dest[x] = 0) THEN
								myRelLineDest[n].dest[x] := myRelLine[n];
							END_IF;
							IF Bag[myBag].Dst = myRelLineDest[n].dest[x] THEN
								myLine := n;
							END_IF;
							IF (myLine > 0)THEN
								EXIT;
							END_IF;
						END_FOR;
						IF (myLine > 0) THEN
							EXIT;
						END_IF;
					END_FOR;
				ELSE
					myLine := alt;
				END_IF;
				//Check data valid
				IF (myLine > 0) AND (myLine <= LOCAL_MAX_DESTS) THEN
					IF (myTransitBag > 0)  AND (myOutBag[myLine] > 0) THEN
						IF bufferClear[myLine] AND (Bag[myOutBag[myLine]].Cat = 0) AND (Bag[myTransitBag].Cat = 0) THEN
							IF (myRelLine[myLine] > 0) THEN
								C[myRelLine[myLine]] := 0;
							END_IF;
							Bag[myTransitBag] := Bag[myBag];
							Bag[myBag] := Bag[0];
							D[900 + mySeq] := step + myLine;
						ELSIF (Bag[myTransitBag].Cat > 0) THEN
							Alarm[mySeq].Name := ALM_BAG_DATA_ERROR;
							Alarm[mySeq].Bag := myTransitBag;
						ELSIF Line[myRelLine[myLine]].Clear THEN
							Alarm[mySeq].Name := ALM_BAG_NOT_SHOWN_ON_SCREEN;
							Alarm[mySeq].Bag := myOutBag[myLine];
						END_IF;
					ELSIF (myOutBag[myLine] > 0) THEN // Don;t use tranit bag.
						IF bufferClear[myLine] AND (Bag[myOutBag[myLine]].Cat = 0) THEN
							IF (myRelLine[myLine] > 0) THEN
								C[myRelLine[myLine]] := 0;
							END_IF;
							D[900 + mySeq] := step + myLine;
						ELSIF Line[myRelLine[myLine]].Clear THEN
							Alarm[mySeq].Name := ALM_BAG_NOT_SHOWN_ON_SCREEN;
							Alarm[mySeq].Bag := myOutBag[myLine];
						END_IF;
					ELSE//Not configured correctly...
						Alarm[mySeq].Name := ALM_GENERAL_SEQUENCE;
					END_IF;
				ELSE
					Alarm[mySeq].Name := ALM_DEST_NOT_VALID;
				END_IF;
			ELSIF (Bag[myBag].Cat = 0) THEN
				Alarm[mySeq].Name := ALM_BAG_DATA_ERROR;
			END_IF;
		ELSE
			//Empty Bag
			RequestRel.PN[myPoint] := 1;
			IF bufferClear[alt] THEN
				IF (myRelLine[alt] > 0) THEN
					C[myRelLine[alt]] := 0;
				END_IF;
				D[900 + mySeq] := step + alt;
			END_IF;
		END_IF;
	ELSIF ((myBag > 0) AND (Bag[myBag].Cat > 0) AND NOT i_bagAtBuffer AND NOT Std.HaltSysZone[myZone]) THEN
		Alarm[mySeq].Name := ALM_BAG_NOT_SETTLED;
	END_IF;
END_IF;

//Select Points AND release bag,NOTE step is greater than OR equal TO 3 so it will be a different step number FOR each destination.
IF (step >= 3) THEN
	myLine := step - 2;
	releaseValid := ((myTransitBag = 0) OR ((Bag[myTransitBag].Cat > 0) AND (Bag[myOutBag[myLine]].Cat = 0)));
	o_select[myLine] :=	TRUE;
	o_openBuffer := releaseValid;
	bagReleased := (((myRelLine[myLine] > 0) AND Line[myRelLine[myLine]].Trip) OR ((myRelLine[myLine] = 0) AND NOT bagArrived[myLine]));
	IF bagReleased AND releaseValid THEN
		IF (myTransitBag > 0) AND (myOutBag[myLine] > 0) AND (myRelLine[myLine] > 0) THEN//Only transfer bag data out when releasing to a buffer.
			Bag[myOutBag[myLine]] := Bag[myTransitBag];
			Bag[myTransitBag] := Bag[0];
		ELSIF (myTransitBag = 0) AND (myOutBag[myLine] > 0) AND (myRelLine[myLine] > 0) THEN//Only transfer bag data out when releasing to a buffer.
			Bag[myOutBag[myLine]] := Bag[myBag];
			Bag[myBag] := Bag[0];
		END_IF;
		IF (myRelLine[myLine] = 0) AND (myBag > 0) THEN // Check data has been deleted by outgoing sequence when tracking bags and using request/enable
			IF (myTransitBag > 0) AND Bag[myTransitBag].Cat = 0 THEN
				D[900 + mySeq]  := 1;
			ELSIF (myOutBag[myLine] > 0) THEN
				IF Bag[myOutBag[myLine]].Cat > 0 THEN
					D[900 + mySeq]  := 1;
				END_IF;
			ELSE
				Alarm[mySeq].Name := ALM_BAG_DATA_ERROR;
			END_IF;
		ELSE
			D[900 + mySeq]  := 1;
		END_IF;
	ELSIF NOT releaseValid THEN
		IF Bag[myTransitBag].Cat = 0 THEN
			Alarm[mySeq].Name := ALM_BAG_DATA_ERROR;
		ELSIF Line[myRelLine[myLine]].Clear AND (Bag[myOutBag[myLine]].Cat > 0) THEN
			Alarm[mySeq].Name := ALM_BAG_DATA_ERROR;
			Alarm[mySeq].Bag := myOutBag[myLine];
		END_IF;
	END_IF;
END_IF;

//-----------------------------------
//PLC Outputs - adjust TO suit system
//-----------------------------------

Y[myIO].Y06 := o_openBuffer;
//EnableRel.IC[1] := o_openBuffer;// Example of using RequestRel interface.

Y[myIO].Y07 := o_select[1];
Y[myIO].Y08 := o_reset OR o_select[2];

//Alarms
timerAlarm(IN := NOT pls AND (Alarm[mySeq].Name > 0),PT:= Alarm[mySeq].Time);

Alarm[mySeq].On 	:= timerAlarm.Q;
Alarm[mySeq].ET 	:= timerAlarm.ET;

END_PROGRAM
```

#### _httpRequest.st
```iecst
ACTION _httpRequest:

	CASE HTTP_Comm[myHttp].Status OF

		HTTP_COMM_STATUS_DISABLED:
			//Build Request String..
			itoa(myBagNumber,ADR(bagNoString));

			//http://10.8.4.220/maintenance/api/Bags/bagCountUpdate?bagNumber=1&plcStation=0

			requestURL := HTTP_POST_MAINT_BAGCOUNT;
			requestURL := CONCAT(requestURL,'plcStation=');
			requestURL := CONCAT(requestURL,Std.PLCStnString);
			requestURL := CONCAT(requestURL,'&bagNumber=');
			requestURL := CONCAT(requestURL,bagNoString);

			requestData := 'FIX ME I SHOULDN T NEED TO BE HERE';

			HTTP_Comm[myHttp].Command.Method := httpMETHOD_POST;//Should httpMethod_POST
			HTTP_Comm[myHttp].Command.Cmd_URL := requestURL;
			HTTP_Comm[myHttp].Command.Body_Data.Adr := ADR(requestData);
			HTTP_Comm[myHttp].Command.Body_Data.Size := strlen(ADR(requestData));
			HTTP_Comm[myHttp].Command.ResponseData.Adr := ADR(httpResponse);
			HTTP_Comm[myHttp].Command.ResponseData.Size := SIZEOF(httpResponse);

			HTTP_Comm[myHttp].Status := HTTP_COMM_STATUS_ACTIVE_WAIT_BUF;

		HTTP_COMM_STATUS_ACTIVE_WAIT_BUF:
			//Command is sent to ring buffer.
		HTTP_COMM_STATUS_IN_BUFFER:
			//Command recieved and in ring buffer
		HTTP_COMM_STATUS_IN_PROCESS:
			//Command being processed by httpClient.
		HTTP_COMM_STATUS_COMPLETE:
			//Decode response Data.
			//The response comes as string... In this case it is easier to read from the byte direct as the response is limited in the SQL proc.
			Bag[myBag].Ur1 := myBagNumber;
			Bag[myBag].Ur2 := UDINT_TO_UINT(atoi(ADR(httpResponse))); //Maintenance State
			IF (Bag[myBag].Ur2 > 0) THEN
				Bag[myBag].Ur2 := (Bag[myBag].Ur2 - 1);
			END_IF;

			//verificationState := UDINT_TO_UINT(atoi(ADR(httpResponse[3]))); // Batch Verification State
			//httpComplete := 1;
			HTTP_Comm[myHttp].Status := HTTP_COMM_STATUS_DISABLED;

		HTTP_COMM_STATUS_ERROR:
			IF (myBagNumber > 0) THEN
				Bag[myBag].Ur1 := myBagNumber;
			ELSE
				Bag[myBag].Ur1 := DEFAULT_BAGNUMBER;
			END_IF;
				HTTP_Comm[myHttp].Status := HTTP_COMM_STATUS_DISABLED;

	END_CASE;

END_ACTION
```

### Program Logical/MaintenancePackage/zzWriteSeqCount (IEC) - *Collect and write Sequence Counts

#### zzWriteSeqCount.ab - Implementation code
```automation-basic
(********************************************************************
 * COPYRIGHT -- HP
 ********************************************************************
 * Program: zzWriteSeqCount
 * File: zzWriteSeqCount.ab
 * Author: treamsbottom
 * Created: October 02, 2013
 ********************************************************************
 * Implementation of program zzWriteSeqCount
 ********************************************************************)

PROGRAM _INIT

END_PROGRAM

PROGRAM _CYCLIC

mySql = 99

//Collect Data
LOOP n = 1  TO Std.MaxSeq DO
	IF (D[900 + n] = 1) AND NOT Index[n] THEN
		Index[n]= TRUE;
		Count[n] = Count[n] + 1;
	ELSE IF (D[900 + n] > 1) THEN
		Index[n] = FALSE;
	ENDIF;
ENDLOOP

LOOP n = 1 TO Std.MaxSeq DO
	IF (Count[n] > 0) AND NOT SqlWriteActive THEN ; Write Count to SQL
		SqlWriteActive = TRUE
		SqlWriteIndex = n
		SqlRequest[mySql].Request = TRUE
		itoa(SqlWriteIndex,ADR(mySeqNum))
		itoa(Count[SqlWriteIndex],ADR(myCount))
		Count[SqlWriteIndex] = 0 ; Reset Count
		SqlRequest[mySql].SQLType = cSQLType_WriteOnly
		SqlRequest[mySql].SQL_usp = cSQLReq_WriteSeqCount
		SqlRequest[mySql].NoOfParams = 3

		SqlRequest[mySql].Parameters[0].Type = cSQLParam_Input
		strcpy(ADR(SqlRequest[mySql].Parameters[0].Param_String),ADR(Std.PLCStnString))
		SqlRequest[mySql].Parameters[1].Type = cSQLParam_Input
		strcpy(ADR(SqlRequest[mySql].Parameters[1].Param_String),ADR(mySeqNum))
		SqlRequest[mySql].Parameters[2].Type = cSQLParam_Input
		strcpy(ADR(SqlRequest[mySql].Parameters[2].Param_String),ADR(myCount))
	ENDIF
EXITIF SqlWriteActive AND (SqlWriteIndex > 0)
ENDLOOP

IF SqlRequest[mySql].Complete THEN ; ClearRequest
	SqlRequest[mySql] = cEmptySQlReq
	SqlWriteActive = FALSE
ENDIF

END_PROGRAM
```

#### zzWriteSeqCount.var - Local variables
```iecst
(********************************************************************
 * COPYRIGHT -- HP
 ********************************************************************
 * Program: zzWriteSeqCount
 * File: zzWriteSeqCount.var
 * Author: treamsbottom
 * Created: October 02, 2013
 ********************************************************************
 * Local variables of program zzWriteSeqCount
 ********************************************************************)
VAR
	Index : ARRAY[0..99] OF BOOL;
	SqlWriteActive : BOOL;
	mySqlreqIndex : INT;
	mySql : UINT;
	myPLCStn : STRING[1];
	SqlWriteIndex : UINT;
	mySeqNum : STRING[5];
	myCount : STRING[10];
	TestTim : BOOL;
	n : UINT;
END_VAR
```

### Request_Constants.var
```iecst
VAR CONSTANT
	HTTP_IF_CALL_USP_NOREPLY_URL : STRING[100] := '/httpcomms/api/plcToSql/calluspnoquery'; (**POST Put Procedure string in the body data*)
	HTTP_IF_CALL_USP_REPLY_URL : STRING[100] := '/httpcomms/api/plcToSql/callusp?sql='; (**GET Function - Put Procedure in URL*)
END_VAR
(*POST - USPS*)
VAR CONSTANT
	HTTP_POST_MAINT_COMPLETE : STRING[100] := '[SUPDB].[Maintenance].[uspMaintenanceBagMaintComplete]'; (*Maint Complete. Needs @PLC,@Bag*)
	HTTP_USP_WRITE_SEQ_COUNT_DATA : STRING[100] := '[SUPDB].[PLC].[uspWriteSequenceCount]'; (*Stored procedure uspWriteSequenceCount. Requires @PLCStn, @SeqNum, @CountIn*)
	HTTP_USP_WRITE_REPORT_DATA : STRING[100] := '[SUPDB].[PLC].[uspReportWrite]'; (*Stored procedure uspReportWrite*)
	HTTP_POST_BATCH_LOCATION_UPDATE : STRING[100] := '[SUPDB].[Master].[uspBatch_LocationUpdate]'; (*Stored procedure [Master].[uspBatch_LocationUpdate] Update batch location.
*)
	HTTP_POST_BATCH_PROPERTY_UPDATE : STRING[100] := '[SUPDB].[Master].[uspBatch_Property_Update]'; (*Stored procedure [Master].[uspBatch_Property_Update] Update a single batch propery by name...
*)
END_VAR
(*GET*)
VAR CONSTANT
	HTTP_GET_SUPERTRACK_CON_STATUS : STRING[100] := '/supertrack/api/settings/connectOpc';
	HTTP_GET_OPCUA_CONNECTION_STATUS : STRING[100] := '/KanDisplay.Manager.API/api/settings/connectOpc';
	HTTP_GET_MAINT_COMPLETE : STRING[100] := '[SUPDB].[Maintenance].[uspMaintenanceBagMaintComplete]'; (*Maint Complete. Needs @PLC,@Bag*)
	HTTP_GET_MAINT_COUNT_REPLY_STATE : STRING[100] := '[SUPDB].[Maintenance].[uspMaintenanceBagCountReplyState]'; (*Send count value, reply state. Needs @PLC,@Bag, @State OUTPUT>.*)
	HTTP_GET_BATCH_CREATE_LOC_UPDATE : STRING[100] := '[SUPDB].[Master].[uspBatch_Create_UpdateLocation]'; (*Update batch location, or create batch if it doesn't exist.*)
END_VAR
(*MIS Batch Interface ADRETT SPECIAL*)
VAR CONSTANT
	HTTP_GET_BATCH_CREATE : STRING[100] := '[SUPDB].[PLC].[uspMIS_BatchCreate]'; (*Update batch location, or create batch if it doesn't exist.*)
END_VAR
```

### Server_Functions.var
```iecst
VAR CONSTANT
	HTTP_SVR_FNC_NOT_FOUND : UINT := 0;
	HTTP_SVR_GET_FNC_IOLINK : UINT := 3;
	HTTP_SVR_GET_FNC_RESTART_PLC : UINT := 4;
	HTTP_SVR_GET_FNC_SET_BAG_DEST : UINT := 1;
	HTTP_SVR_GET_FNC_TEST : UINT := 2;
	HTTP_SVR_POST_FNC_IOLINK : UINT := 30;
	HTTP_SVR_POST_FNC_TEST : UINT := 20;
	HTTP_SVR_GET_FNC_IOLINK_STATUS : UINT := 6;
	HTTP_SVR_GET_FNC_IOLINK_GEN_FILE : UINT := 5;
	HTTP_SVR_POST_FNC_ABB : UINT := 70;
	HTTP_SVR_GET_FNC_ABB : UINT := 7;
END_VAR
```

### Variables.var
```iecst
VAR CONSTANT
	HTTP_MAX_COMM : UINT := 20; (**Max number of interfaces to talk to http.*)
END_VAR
VAR
	HTTP_Comm : ARRAY[0..HTTP_MAX_COMM] OF http_comm_typ;
	HTTP_Config : httpConfig_typ;
END_VAR
```

### Types.typ - Exported data types
```iecst
TYPE
	http_comm_typ : 	STRUCT
		Command : http_Cmd_typ; (**Set the values to pass into the http comm driver,*)
		Status : HTTP_Status_enum; (**Status of the http comm driver.*)
		LastError : STRING[60]; (**String to describe the last error*)
		lastResponse : httpResponseHeader_t;
	END_STRUCT;
	http_Cmd_typ : 	STRUCT
		Method : UINT; (*Set the http cmd type.. POST,GET,PUT,DELETE*)
		Cmd_URL : STRING[254]; (*The string data appended to the URL - Use with GET and DELETE *)
		Body_Data : dataPointer_typ; (*Data to send in the body of the message - USE with POST and PUT*)
		ResponseData : dataPointer_typ; (*Data address of where to set the http response data*)
	END_STRUCT;
	dataPointer_typ : 	STRUCT
		Adr : UDINT;
		Size : UDINT;
	END_STRUCT;
	HTTP_Status_enum :
		(
		HTTP_COMM_STATUS_DISABLED,
		HTTP_COMM_STATUS_ACTIVE_WAIT_BUF,
		HTTP_COMM_STATUS_IN_BUFFER,
		HTTP_COMM_STATUS_IN_PROCESS,
		HTTP_COMM_STATUS_COMPLETE,
		HTTP_COMM_STATUS_ERROR
		);
	httpConfig_typ : 	STRUCT
		Host : STRING[20];
		Port : UINT;
	END_STRUCT;
END_TYPE
```

### Program Logical/http_Lib/zzHttpDriver (IEC, version 1.01.0)

#### Variables.var - Local variables
```iecst
VAR
	n : UINT;
	r : UINT;
	httpComm : REFERENCE TO http_comm_typ;
	ringBuffer : ARRAY[0..HTTP_MAX_COMM] OF UINT;
	sizeRingArray : UDINT;
	sizeRingData : UDINT;
	moveSize : UDINT;
	pUrl : UDINT;
	URL : STRING[280];
	pHost : UDINT;
	pResponseHeader : UDINT;
	pTempMem : UDINT;
	sizeTempMem : UDINT;
	pStatistics : UDINT;
	responseHeader : httpResponseHeader_t;
	http_Client : httpClient;
	Statistics : httpStatistics_t;
	emptyResponseHeader : httpResponseHeader_t;
	abort : BOOL;
	DebugErrCount : UDINT;
	pRequestHeader : UDINT;
	requestHeader : httpRequestHeader_t;
	debugToUSB : BOOL;
	fileRW : fileReadWrite;
	errorData : STRING[1000];
	remainingStringLen : DINT;
END_VAR
```

#### Main.st - Init, cyclic, exit code
```iecst
PROGRAM _INIT
	//Use Static code now but change to config file later..
	HTTP_Config.Host := '10.8.4.220';
	HTTP_Config.Port := 0;

	//Configure RequestHeader
	requestHeader.protocol := 'HTTP/1.1';
	requestHeader.host := HTTP_Config.Host;
	requestHeader.contentType := 'text/plain';
	requestHeader.connection := 'Keep-Alive';
	requestHeader.keepAlive := 'max=100,timeout=5';
	//Turn off Debug.
	debugToUSB := 0;

	pHost := ADR(requestHeader.host);
	pUrl := ADR(URL);
	pRequestHeader := ADR(requestHeader);
	pResponseHeader := ADR(responseHeader);
	pStatistics := ADR(Statistics);
	sizeTempMem := 5000000; //Allocate 5MB of free memory
	TMP_alloc(sizeTempMem,ADR(pTempMem));
	//Check for any requests that were being processed on shut down..
	FOR n := 1 TO HTTP_MAX_COMM DO
		IF HTTP_Comm[n].Status = HTTP_COMM_STATUS_IN_PROCESS THEN
			ringBuffer[0] := n;
		ELSIF HTTP_Comm[n].Status = HTTP_COMM_STATUS_IN_BUFFER THEN
			ringBuffer[n] := n;
		END_IF;
	END_FOR;
	_orderRing;
END_PROGRAM

PROGRAM _CYCLIC

	//Listen to requests and add to ring buffer.
	_ringBuffer;

	//For this mod to work, we have to remove the dynamic ref to httpComm in _ringBuffer adn _addToRing
	//Wait for next command from ring buffer
	IF (ringBuffer[0] = 0) AND (ringBuffer[1] > 0) THEN
		ringBuffer[0] := ringBuffer[1];
		httpComm ACCESS ADR(HTTP_Comm[ringBuffer[0]]);
		httpComm.Status := HTTP_COMM_STATUS_IN_PROCESS;
	ELSIF (ringBuffer[0] > 0) THEN
		httpComm ACCESS ADR(HTTP_Comm[ringBuffer[0]]);
	END_IF;

	httpComm ACCESS ADR(HTTP_Comm[ringBuffer[0]]);
//	IF (ringBuffer[0] > 0) THEN
//		httpComm.Status := HTTP_COMM_STATUS_IN_PROCESS;
//	END_IF

	//Call the Http fub.
	_httpComm;
END_PROGRAM
```

#### _httpComm.st
```iecst
//HTTP Client function...
//Read all requests into temporary memory.
ACTION _httpComm:
	//Build URL
	URL := httpComm.Command.Cmd_URL;

	requestHeader.contentLength := httpComm.Command.Body_Data.Size;

	http_Client.enable := 1;
	http_Client.send := ((httpComm.Status = HTTP_COMM_STATUS_IN_PROCESS) AND NOT abort);
	http_Client.abort := abort;
	http_Client.option := httpOPTION_HTTP_11;
	http_Client.pHost := pHost;
	http_Client.hostPort := HTTP_Config.Port;
	http_Client.pUri := pUrl;
	http_Client.pRequestHeader := pRequestHeader;
	http_Client.method := httpComm.Command.Method;
	http_Client.pRequestData := httpComm.Command.Body_Data.Adr;
	http_Client.requestDataLen := httpComm.Command.Body_Data.Size;
	http_Client.pResponseHeader := pResponseHeader;
	http_Client.pResponseData := pTempMem;
	http_Client.responseDataSize := sizeTempMem;
	http_Client.pStatistics := pStatistics;
	//http_Client();

	IF (http_Client.status = ERR_OK) THEN
		abort := 0;
//		IF http_Client.tcpStatus = tcpERR_NOT_CONNECTED THEN
//			abort := 1;
//			httpComm.Status := HTTP_COMM_STATUS_ERROR;
//			ELS
		IF (httpComm.Status = HTTP_COMM_STATUS_IN_PROCESS) THEN;
			IF (responseHeader.status = '200 OK') THEN
				IF (responseHeader.contentLength > 0) THEN
					IF (responseHeader.contentLength <= httpComm.Command.ResponseData.Size) THEN
						memset(httpComm.Command.ResponseData.Adr,0,httpComm.Command.ResponseData.Size);
						memmove(httpComm.Command.ResponseData.Adr,pTempMem,responseHeader.contentLength);
						httpComm.Status := HTTP_COMM_STATUS_COMPLETE;
					ELSE
						httpComm.Status := HTTP_COMM_STATUS_ERROR;
						httpComm.LastError := 'Response data area to small';
					END_IF;
				ELSIF (httpComm.Command.Method = httpMETHOD_POST) THEN
					httpComm.Status := HTTP_COMM_STATUS_COMPLETE;
				END_IF;
			ELSIF (responseHeader.status <> emptyResponseHeader.status) THEN
				IF debugToUSB THEN
					//Build Debug Data.
					strcpy(ADR(errorData),ADR(''));
					//memcpy(ADR(errorData),pTempMem,SIZEOF(errorData));//,responseHeader.contentLength);

					strcpy(ADR(errorData),ADR('Request Header - '));
					strcat(ADR(errorData),pRequestHeader);
					strcat(ADR(errorData),ADR('$r$n'));
					strcat(ADR(errorData),ADR('Request URL - '));
					strcat(ADR(errorData),pUrl);
					strcat(ADR(errorData),ADR('$r$n'));

					strcat(ADR(errorData),ADR('Request Body - '));
					IF httpComm.Command.Body_Data.Adr > 0 THEN
						strcat(ADR(errorData),httpComm.Command.Body_Data.Adr);
					ELSE
						strcat(ADR(errorData),ADR('no body sent'));
					END_IF;
					strcat(ADR(errorData),ADR('$r$n'));
					strcat(ADR(errorData),ADR('Response Data :'));
					strcat(ADR(errorData),ADR('$r$n'));
					//Check message will fit in error string.
					remainingStringLen := SIZEOF(errorData) - LEN(errorData) - 5; //Subtract extra 5 to make room for end of line characters
					IF (strlen(pTempMem) <= remainingStringLen) THEN
						strcat(ADR(errorData), pTempMem);
					ELSE
						strcat(ADR(errorData),ADR('Response message to large use postman'));
					END_IF;
					strcat(ADR(errorData),ADR('$r$n'));

					fileRW.enable := 1;
					fileRW.mode := FILE_SAVE;
					fileRW.pFileDevice := ADR('USBStick');
					fileRW.pFileName := ADR('HttpError.txt') ;//adrFileName;
					fileRW.pData := ADR(errorData);
					fileRW.sizeData := strlen(ADR(errorData));
					fileRW.appendToFile := 1;
					fileRW();
					IF fileRW.status = ERR_OK THEN
						httpComm.Status := HTTP_COMM_STATUS_ERROR;
						httpComm.LastError := responseHeader.status;
						//debugToUSB := FALSE;
					ELSIF fileRW.status <> ERR_FUB_BUSY THEN
						httpComm.Status := HTTP_COMM_STATUS_ERROR;
						httpComm.LastError := responseHeader.status;
					END_IF;
				ELSE
					httpComm.Status := HTTP_COMM_STATUS_ERROR;
					httpComm.LastError := responseHeader.status;
				END_IF;
			ELSIF (responseHeader.status = emptyResponseHeader.status) THEN
//				httpComm.Status := HTTP_COMM_STATUS_ERROR;
//				httpComm.LastError := responseHeader.status;
//				abort := 1;
			END_IF;
		END_IF;
		//The B&R function block does not return status 0, when there is no data in the reponse body and we use the GET method.
	ELSIF ((http_Client.status = ERR_FUB_BUSY) AND (responseHeader.status = '200 OK') AND (httpComm.Command.ResponseData.Size = 0))THEN // AND (httpComm.Command.Method = httpMETHOD_GET)) THEN // THere is no data to recieve so the fub will not complete.
		httpComm.Status := HTTP_COMM_STATUS_COMPLETE;
		httpComm.LastError := 'Wrong method used- USE POST with no response data';
		http_Client.enable := 0;
	ELSIF (http_Client.status = httpERR_BUFFER_SIZE) THEN
		httpComm.Status := HTTP_COMM_STATUS_ERROR;
		httpComm.LastError := 'temp data area to small';
	ELSIF (http_Client.status <> ERR_FUB_BUSY) THEN
		DebugErrCount := DebugErrCount + 1;
		itoa(http_Client.status,ADR(httpComm.LastError));
		abort := 1;
	END_IF;
	//We make sure we turn of the http send command between requests..
	IF EDGEPOS(httpComm.Status <> HTTP_COMM_STATUS_IN_PROCESS) THEN
		http_Client.send := 0;
		//http_Client();
		httpComm.lastResponse := responseHeader;
		ringBuffer[0] := 0;//Clear the comm object from the active part of ring buffer
		responseHeader := emptyResponseHeader;
		//memset(pTempMem,0,sizeTempMem); Giving cycle time errors.. There is no need to clear this memory anyway as we only copy the reposonse length.
	END_IF;
	http_Client();
END_ACTION
```

### Library Logical/http_Lib/KanHttp (IEC)

#### KanHttp.fun - Exported functions and function blocks
```iecst
FUNCTION_BLOCK httpGetParameter (*FUB to Get parameter values set in URI or BODY...*) (*$GROUP=User,$CAT=User,$GROUPICON=User.png,$CATICON=User.png*)
	VAR_INPUT
		searchPropertyName : STRING[50]; (*StringValue of propery or name to match*)
		searchEndProperty : STRING[50]; (*String Character or value to show end of property value -- DEFAULT & *)
		searchOffset : UINT; (*Offset can be set to skip searching begining of string if not required*)
		searchString : {REDUND_UNREPLICABLE} STRING[5000];
	END_VAR
	VAR_OUTPUT
		outputValue : STRING[100]; (*String Value found*)
		status : UINT;
		postionFound : UINT; (*Start position of the data found *)
	END_VAR
	VAR
		matchString : STRING[50];
		inputData : ARRAY[0..4999] OF USINT;
		endIndex : UINT;
		startPosition : UINT;
		n : UINT;
		compare : DINT;
		length : UINT;
		startoffset : UINT;
		search : STRING[50];
	END_VAR
END_FUNCTION_BLOCK
```

### Program Logical/http_Lib/httpServer (IEC) - *Listen for http requests

#### Variables.var - Local variables
```iecst
VAR
	httpServer : httpService;
	sendResponse : BOOL;
	abortResponse : BOOL;
	URI : STRING[500];
	requestHeader : httpRequestHeader_t;
	requestData : STRING[10000];
	responseHeader : httpResponseHeader_t;
	responseData : STRING[10000];
	Statistics : httpStatistics_t;
	serviceName : STRING[50];
	getParameterName : httpGetParameter;
END_VAR
VAR CONSTANT
	STRING_DOLLAR : STRING[1] := '&';
END_VAR
VAR
	activeFunction : UINT;
	mis : UDINT;
	bagIndex : UDINT;
	dst : USINT;
	error : INT;
END_VAR
```

#### Main.st - Init, cyclic, exit code
```iecst
PROGRAM _INIT
	serviceName := 'supertrackPLC.api';
	httpServer.pServiceName := ADR(serviceName);
	httpServer.pUri := ADR(URI);
	httpServer.uriSize := SIZEOF(URI);
	httpServer.pRequestHeader := ADR(requestHeader);
	httpServer.pRequestData := ADR(requestData);
	httpServer.requestDataSize := SIZEOF(requestData);
	httpServer.pResponseHeader := ADR(responseHeader);
	httpServer.pResponseData := ADR(responseData);

	httpServer.pStatistics := ADR(Statistics);

	httpServer.option := httpOPTION_HTTP_11 + httpOPTION_SERVICE_TYPE_NAME; //HTTP 1.1

END_PROGRAM

PROGRAM _CYCLIC

	httpServer.enable := 1;
	httpServer.send := sendResponse; // Send Response on Rising edge.
	httpServer.abort := abortResponse;	//Send abort Response on Rising Edge
	httpServer();

	sendResponse := 0;
	abortResponse := 0;

	IF httpServer.status = ERR_OK THEN
	//Get The Function Name --		1
		IF activeFunction = 0 THEN _getFunctionName; END_IF;
	//Exectute the Function
		CASE activeFunction OF
			HTTP_SVR_FNC_NOT_FOUND: //Nothing
				sendResponse := 1;
				memset(ADR(responseData),0,SIZEOF(responseData));//Clear responseData
				responseData := 'error Function Not found, Function Must be specified with function=';
				httpServer.responseDataLen := LEN(responseData);

			HTTP_SVR_GET_FNC_SET_BAG_DEST: //Set Bag Destination -- 1
//				_setBagDestination;
			HTTP_SVR_GET_FNC_TEST://Test
				sendResponse := 1;
				memset(ADR(responseData),0,SIZEOF(responseData));//Clear responseData
				responseData := 'Test Get';
				httpServer.responseDataLen := LEN(responseData);

//			HTTP_SVR_GET_FNC_IOLINK://IO_Link GET function
//				sendResponse := 1;
//				memset(ADR(responseData),0,SIZEOF(responseData));//Clear responseData
//				responseData := IO_Link.httpResponse;
//				httpServer.responseDataLen := LEN(responseData);
//				IO_Link.Load := TRUE; //Reload httpResponse with XML data incase its a after status http call

			HTTP_SVR_GET_FNC_RESTART_PLC:
				sendResponse := 1;
				memset(ADR(responseData),0,SIZEOF(responseData));//Clear responseData
				responseData := 'PLC will carry out a warm restart';
				httpServer.responseDataLen := LEN(responseData);
				IF httpServer.phase = 4 THEN //Wait for response to be sent
					SYSreset(TRUE,1); //Restart PLC
				END_IF;

//			HTTP_SVR_GET_FNC_IOLINK_GEN_FILE://IO_Link GET function Generate file
//				sendResponse := 1;
//				memset(ADR(responseData),0,SIZEOF(responseData));//Clear responseData
//				responseData := 'Config File Generated';
//				httpServer.responseDataLen := LEN(responseData);
//				IO_Link.Save := TRUE;

//			HTTP_SVR_GET_FNC_IOLINK_STATUS://IO_Link GET function Status request
//				sendResponse := 1;
//				memset(ADR(responseData),0,SIZEOF(responseData));//Clear responseData
//				responseData := 'Status Loaded';
//				httpServer.responseDataLen := LEN(responseData);
//				IO_Link.Status := TRUE;

			HTTP_SVR_GET_FNC_ABB://ABB GET function Status request
					sendResponse := 1;
					memset(ADR(responseData),0,SIZEOF(responseData));//Clear responseData
					responseData := ABB_EPL.httpRequest;
					httpServer.responseDataLen := LEN(responseData);

//			HTTP_SVR_POST_FNC_IOLINK://IO_Link POST function
//				sendResponse := 1;
//				memset(ADR(responseData),0,SIZEOF(responseData));//Clear responseData
//				responseData := 'IOLinkPost';
//				httpServer.responseDataLen := LEN(responseData);
//				//Clear IO_Link.httpResponse if file found
//				memset(ADR(IO_Link.httpResponse),0,SIZEOF(IO_Link.httpResponse));
//				IO_Link.httpResponse := requestData;
//				IO_Link.httpRequestState := 1;

			HTTP_SVR_POST_FNC_ABB://IO_Link POST function
					sendResponse := 1;
					memset(ADR(responseData),0,SIZEOF(responseData));//Clear responseData
					responseData := 'ABBPost';
					httpServer.responseDataLen := LEN(responseData);
					//Clear ABB_EPL.httpResponse
					memset(ADR(ABB_EPL.httpResponse),0,SIZEOF(ABB_EPL.httpResponse));
					memcpy(ADR(ABB_EPL.httpResponse),ADR(requestData),SIZEOF(ABB_EPL.httpResponse));
					ABB_EPL.callBackUpWrite := TRUE;

		END_CASE
	ELSE
		activeFunction := 0;
	END_IF;

END_PROGRAM

PROGRAM _EXIT
	//Disable the Server on Exit..
	httpServer.enable := 1;
	httpServer();
END_PROGRAM
```

#### _getFunctionName.st
```iecst
ACTION _getFunctionName:
	CASE httpServer.method OF
		httpMETHOD_DELETE,httpMETHOD_PUT:
			//wrong method-- implement error handling.

		httpMETHOD_GET:
			getParameterName.searchString := URI;
			getParameterName.searchOffset := LEN(serviceName);
		httpMETHOD_POST:
			getParameterName.searchString := URI;
			getParameterName.searchOffset := LEN(serviceName);
//			getParameterName.searchString := requestData;
//			getParameterName.searchOffset := 0;
	END_CASE;

	getParameterName.searchPropertyName := 'function=';
	getParameterName.searchEndProperty := STRING_DOLLAR ;
	getParameterName();

	CASE httpServer.method OF
		httpMETHOD_DELETE,httpMETHOD_PUT:
			//wrong method-- implement error handling.

		httpMETHOD_GET:
			IF getParameterName.status = ERR_OK THEN
				IF getParameterName.outputValue = 'dmSetDst' THEN activeFunction := HTTP_SVR_GET_FNC_SET_BAG_DEST;
				ELSIF getParameterName.outputValue = 'test' THEN activeFunction := HTTP_SVR_GET_FNC_TEST;
//				ELSIF getParameterName.outputValue = 'iolink' THEN activeFunction := HTTP_SVR_GET_FNC_IOLINK;
				ELSIF getParameterName.outputValue = 'restart' THEN activeFunction := HTTP_SVR_GET_FNC_RESTART_PLC;
//				ELSIF getParameterName.outputValue = 'iolinkGenFile' THEN activeFunction := HTTP_SVR_GET_FNC_IOLINK_GEN_FILE;
//				ELSIF getParameterName.outputValue = 'iolinkStatus' THEN activeFunction := HTTP_SVR_GET_FNC_IOLINK_STATUS;
				ELSIF getParameterName.outputValue = 'ABB' THEN activeFunction := HTTP_SVR_GET_FNC_ABB;
				ELSE activeFunction := HTTP_SVR_FNC_NOT_FOUND;
				END_IF;
				getParameterName.searchString := '';
			END_IF;
		httpMETHOD_POST:
			IF getParameterName.status = ERR_OK THEN
				IF getParameterName.outputValue = 'test' THEN activeFunction := HTTP_SVR_POST_FNC_TEST;
//				ELSIF getParameterName.outputValue = 'iolink' THEN activeFunction := HTTP_SVR_POST_FNC_IOLINK;
				ELSIF getParameterName.outputValue = 'ABB' THEN activeFunction := HTTP_SVR_POST_FNC_ABB;
				ELSE activeFunction := HTTP_SVR_FNC_NOT_FOUND;
				END_IF;
				getParameterName.searchString := '';
			END_IF;
	END_CASE;

END_ACTION
```

#### LocalFunctions.fun
```iecst
FUNCTION_BLOCK httpGetParameter (*FUB to Get parameter values set in URI or BODY...*) (*$GROUP=User,$CAT=User,$GROUPICON=User.png,$CATICON=User.png*)
	VAR_INPUT
		searchPropertyName : STRING[50]; (*StringValue of propery or name to match*)
		searchEndProperty : STRING[50]; (*String Character or value to show end of property value -- DEFAULT & *)
		searchOffset : UINT; (*Offset can be set to skip searching begining of string if not required*)
		searchString : STRING[500];
	END_VAR
	VAR_OUTPUT
		outputValue : STRING[100]; (*String Value found*)
		status : UINT;
	END_VAR
	VAR
		matchString : STRING[50];
		inputData : ARRAY[0..499] OF USINT;
		endIndex : INT;
		startPosition : INT;
		n : INT;
		compare : DINT;
		length : UINT;
		startoffset : UINT;
		search : STRING[50];
	END_VAR
END_FUNCTION_BLOCK
```

#### httpGetParameter.st
```iecst
(* FUB to Get parameter values set in URI or BODY... *)
FUNCTION_BLOCK httpGetParameter
	status := ERR_FUB_BUSY;
// Get the function Name from the URI
//Use the string length of the service name	+
	memset(ADR(outputValue),0,SIZEOF(outputValue));
	matchString := searchPropertyName;
	strcpy(ADR(inputData[0]),ADR(searchString));
	startoffset := searchOffset;
	endIndex := LEN(searchString);
	startPosition := 16#FFF;
	IF endIndex > startoffset THEN
		FOR n := startoffset TO endIndex DO
			memcpy(ADR(search),ADR(inputData[n]),LEN(matchString));
			compare := 	strcmp(ADR(search),ADR(matchString));
			IF (compare = 0) THEN
				startPosition := n + LEN(matchString);
				EXIT;
			END_IF;
		END_FOR;
	ELSE
		status := 100;
	END_IF;

	IF (startPosition <> 16#FFF) THEN
		//Get the End Position
		matchString := searchEndProperty;
		memset(ADR(search),0,SIZEOF(search));
		startoffset := startPosition;
		IF endIndex >= startoffset THEN
			FOR n := startoffset TO endIndex DO
				memcpy(ADR(search),ADR(inputData[n]),LEN(matchString));
				compare := 	strcmp(ADR(search),ADR(matchString));
				length := n - startPosition;
				IF (compare = 0) THEN
					EXIT;
				END_IF;
			END_FOR;
			outputValue := MID(searchString,length,startPosition + 1);
			status := ERR_OK;
		ELSE
			status := 102;
		END_IF;
	ELSE
		outputValue := '';
		status := 101;
	END_IF;

END_FUNCTION_BLOCK
```

### Library Logical/File_System/FileMgr (IEC)
Depends on: FileIO, DataObj, AsHttp

#### Types.typ - Exported data types
```iecst
TYPE
	fileToDatObj_state :
		(
		Fi_To_Do_INIT,
		Fi_To_Do_FILE_OPEN,
		Fi_To_Do_FILE_READ,
		Fi_To_Do_FILE_CLOSE,
		Fi_To_Do_DObj_GET_INFO,
		Fi_To_Do_DObj_DELETE,
		Fi_To_Do_DObj_CREATE,
		Fi_To_Do_ERROR,
		Fi_To_Do_DObj_WRITE
		);
	fileToMem_state :
		(
		Fi_To_Mem_INIT,
		Fi_To_Mem_FILE_OPEN,
		Fi_To_Mem_FILE_READ,
		Fi_To_Mem_FILE_CLOSE,
		Fi_To_Mem_ERROR
		);
	fileCopyFromDev_state :
		(
		FiCopyDev_INIT,
		FiCopyDev_DEVLINK,
		FiCopyDev_COPY,
		FiCopyDev_UNLINK,
		FiCopyDev_ERROR
		);
	WriteXML_State :
		(
		READY, (**Wait for Pulse of the enable ti start function*)
		CREATE_WRITER,
		START_DOC,
		WRITE_ROOT_ELEMENT,
		READ_DATA_STRUCTURE,
		WRITE_START_ELEMENT,
		WRITE_ELEMENT_TEXT,
		WRITE_END_ELEMENT,
		CLOSE_ALL_ELEMENTS,
		END_DOC,
		CREATE_XML_FILE,
		CLOSE_WRITER,
		FINISHED,
		ERROR
		);
END_TYPE
```

#### FileMgr.fun - Exported functions and function blocks
```iecst
FUNCTION_BLOCK fileReadWrite (**Read or Write to file*) (*$GROUP=User,$CAT=User,$GROUPICON=User.png,$CATICON=User.png*)
	VAR_INPUT
		enable : BOOL;
		pFileDevice : UDINT;
		pFileName : UDINT;
		mode : UINT;
		pData : UDINT; (*point to data to read or write to*)
		sizeData : UDINT; (*size of data to read or write to*)
		Offset : UDINT; (*offset of data to be read or written*)
		appendToFile : BOOL;
	END_VAR
	VAR_OUTPUT
		status : UINT;
	END_VAR
	VAR
		fileState : UINT;
		fileOpen : FileOpen;
		fileCreate : FileCreate;
		fileClose : FileClose;
		error : UINT;
		fileWrite : FileWrite;
		ident : UDINT;
		fileRead : FileRead;
	END_VAR
END_FUNCTION_BLOCK

FUNCTION_BLOCK fileToDatObj (**read from a file into a data object. The data object will be deleted and created the same size as file*) (*$GROUP=User,$CAT=User,$GROUPICON=User.png,$CATICON=User.png*)
	VAR_INPUT
		enable : BOOL; (** Enable*)
		pFileDevice : UDINT; (*pointer to file device*)
		pFileName : UDINT; (*pointer to the file name*)
		pDoName : UDINT; (*pointer to the name of the dataObject to be written to*)
		MemType : USINT;
	END_VAR
	VAR_OUTPUT
		status : UINT;
		do_Ident : UDINT; (*pointer to the ident to the data Object*)
		pDatObjMem : UDINT; (*Pointer to the memory area of the data object written to*)
		fiSize : UDINT;
	END_VAR
	VAR
		fileOpen : FileOpen;
		error : UINT;
		fileRead : FileRead;
		fileClose : FileClose;
		fileState : fileToDatObj_state;
		fi_ident : UDINT;
		do_GetInfo : DatObjInfo;
		do_Delete : DatObjDelete;
		do_Create : DatObjCreate;
		do_Write : DatObjWrite;
	END_VAR
END_FUNCTION_BLOCK

FUNCTION_BLOCK fileToMem (**OpenFileInto memory*) (*$GROUP=User,$CAT=User,$GROUPICON=User.png,$CATICON=User.png*)
	VAR_INPUT
		enable : BOOL; (** Enable*)
		pFileDevice : UDINT; (*pointer to file device*)
		pFileName : UDINT; (*pointer to the file name*)
		pTempMem : UDINT; (**point to the memory area created by TMP_alloc*)
		sizeTempMem : UDINT; (**Size of the temporary memory allocated by TMP_alloc*)
	END_VAR
	VAR_OUTPUT
		status : UINT;
		fiSize : UDINT;
	END_VAR
	VAR
		fileOpen : FileOpen;
		error : UINT;
		fileRead : FileRead;
		fileClose : FileClose;
		fileState : fileToMem_state;
		fi_ident : UDINT;
	END_VAR
END_FUNCTION_BLOCK

FUNCTION_BLOCK FileCopyFromDev (**Copy file from devlink link file device*) (*$GROUP=User,$CAT=User,$GROUPICON=User.png,$CATICON=User.png*)
	VAR_INPUT
		enable : BOOL;
		pFileDevice : UDINT;
		pDevLinkParameter : UDINT;
		pFileName : UDINT;
		pDest : UDINT;
		pDestDev : UDINT;
	END_VAR
	VAR_OUTPUT
		status : UINT;
	END_VAR
	VAR
		fileState : fileCopyFromDev_state;
		error : UINT;
		devLink : DevLink;
		fileCopy : FileCopy;
		devUnlink : DevUnlink;
		devHandle : UDINT;
	END_VAR
END_FUNCTION_BLOCK

FUNCTION_BLOCK WriteXMLFromStructure (*Convert Data structure to XML *) (*$GROUP=User,$CAT=User,$GROUPICON=User.png,$CATICON=User.png*)
	VAR_INPUT
		enable : BOOL;
		pData : UDINT; (*pointer to data area to copy the xml fle*)
		sizeData : UDINT; (*Size of the data area to copy the xml file*)
		pStructName : UDINT;
	END_VAR
	VAR_OUTPUT
		status : UINT;
		LastError : UINT;
	END_VAR
	VAR
		state : WriteXML_State;
		createXMLwriter : xmlCreateMemoryWriter;
		ident : UDINT;
		xmlGetMemInfo : xmlGetMemoryInfo;
		zzEdge00000 : BOOL;
		xmlCloseWriter : xmlCloseMemoryWriter;
		pvStatus : UINT;
		index : UINT;
		pvName : STRING[60];
		taskName : STRING[20];
		xmlWriteElementStart : xmlWriteStartElement;
		openElements : UINT; (*Number of elements to close.*)
		xmlWriteEndElement : xmlWriteEndElement;
		noOfElements : UINT;
		pv_dataLen : UDINT;
		pv_dataType : UDINT;
		pvData : STRING[50];
		pName : UDINT;
		zzEdge00001 : BOOL;
		pvFullName : STRING[100];
		val : UDINT;
		pvGetAdrStatus : UINT;
		pv_Adr : UDINT;
		elementVal : STRING[30];
		xmlWriteElemText : xmlWriteElementText;
		xmlEndDocument : xmlWriteEndDocument;
		xmlStartDocument : xmlWriteStartDocument;
		zzEdge00002 : BOOL;
		pv_tryCount : USINT;
		tempString : STRING[30];
	END_VAR
END_FUNCTION_BLOCK
```

#### WriteXMLFromStructure.st
```iecst
(* Convert Data structure to XML  *)
FUNCTION_BLOCK WriteXMLFromStructure

	IF EDGEPOS(enable) THEN
		state := CREATE_WRITER;
		status := ERR_FUB_BUSY;
		openElements := 0;
		LastError := 0;
		pv_tryCount := 0;
		memcpy(pData,ADR(''),sizeData);
	ELSIF EDGENEG(enable) THEN
		state := CLOSE_WRITER;
	END_IF;

	IF EDGEPOS(state = READ_DATA_STRUCTURE) THEN
		openElements := openElements + 1;
	END_IF;

	CASE state OF
		READY://
			//Wait for rising edge of enable to start.

		CREATE_WRITER://Create the XML writer
			createXMLwriter.enable := 1;
			createXMLwriter();
			IF (createXMLwriter.status = ERR_OK) THEN
				ident := createXMLwriter.ident;
				state := START_DOC;
			ELSE
				state := READY;
				LastError := createXMLwriter.status;
			END_IF;

		START_DOC://Set the header and version number
			xmlStartDocument.enable 		:= 1;
			xmlStartDocument.ident 			:= ident;
			xmlStartDocument.pVersion		:= ADR('1.0');
			xmlStartDocument.pEncoding 		:= ADR('UTF-8');
			xmlStartDocument.pStandalone 	:= 0;
			xmlStartDocument();
			IF (xmlStartDocument.status = ERR_OK) THEN
				state := WRITE_ROOT_ELEMENT;
				index := 0;
			ELSIF (xmlStartDocument.status <> ERR_FUB_BUSY) THEN
				LastError := xmlStartDocument.status;
				state := CLOSE_WRITER;
			END_IF;

		WRITE_ROOT_ELEMENT: //Write the ROOT Element -- This is the name of data structure..
			xmlWriteElementStart.enable := 1;
			xmlWriteElementStart.ident := ident;
			xmlWriteElementStart.pName := pStructName;
			xmlWriteElementStart();
			IF (xmlWriteElementStart.status = ERR_OK) THEN
				pName := pStructName;
				state := READ_DATA_STRUCTURE;
			ELSIF (xmlWriteElementStart.status <> ERR_FUB_BUSY) THEN
				LastError := xmlWriteElementStart.status;
				state := CLOSE_WRITER;
			END_IF;

		READ_DATA_STRUCTURE:// Read from the data structure to get the element names
			//What have to pass in the structure Name..
			// Only pass the structure name -- The code will handle it if it;s global or local
			pvStatus := PV_item(pName,index,ADR(pvName));
			IF (pvStatus = ERR_OK) THEN
				//Build the full var name- for use later.
				brsstrcpy(ADR(pvFullName),pName);
				brsstrcat(ADR(pvFullName),ADR('.'));
				brsstrcat(ADR(pvFullName),ADR(pvName));
				state := WRITE_START_ELEMENT;
			ELSIF (pvStatus = 14710)THEN// ERR_SYS_PV_NOT_FOUND)
				pv_tryCount := (pv_tryCount + 1);
				IF (pv_tryCount > 1) THEN
					//Error PV not found
					LastError := pvStatus;
					state := CLOSE_WRITER;
				ELSE
					//Add the taskname in front of the var to declare it as local.
					ST_name(0,ADR(taskName),0);
					brsstrcat(ADR(taskName),ADR(':'));
					brsstrcat(ADR(taskName),pStructName);
					pName := ADR(taskName);
				END_IF;
			ELSIF pvStatus = 14704 THEN //No more elements
				state := CLOSE_ALL_ELEMENTS;
			ELSIF pvStatus <> ERR_FUB_BUSY THEN
				LastError := pvStatus;
				state := CLOSE_WRITER;
			END_IF;

		WRITE_START_ELEMENT:
			xmlWriteElementStart.enable := 1;
			xmlWriteElementStart.ident := ident;
			xmlWriteElementStart.pName := ADR(pvName);
			xmlWriteElementStart();
			IF (xmlWriteElementStart.status = ERR_OK) THEN
				//Check the PV property to see if has a value we need to write.
				pvStatus := PV_ninfo(ADR(pvFullName),ADR(pv_dataType),ADR(pv_dataLen),ADR(noOfElements));
				IF pvStatus = ERR_OK THEN
					//Get the value here. cast it to string to write into element..
					//get the address of the var.
					pvGetAdrStatus := PV_xgetadr(ADR(pvFullName),ADR(pv_Adr),ADR(pv_dataLen));
					IF pvGetAdrStatus = ERR_OK THEN
//Future... Use the noOfElements to be able to write array values..
						//Set the state here to apply to all-- Overwrite in each action if we don't want to write any element data.
						val := 0;
						state := WRITE_ELEMENT_TEXT;
						elementVal := 'Test';
						CASE pv_dataType OF
							0://Structures.. No data for the element
								state := READ_DATA_STRUCTURE;
								index := index + 1;

							1,2,3,4,5,6,7,8,17,18,19,21: //max 32bit data...
								brsmemcpy(ADR(val),pv_Adr,pv_dataLen);
								brsitoa(val,ADR(elementVal));
							9://String
								//Check MAX element text here... 30charss

							10://64Bit numbers ULINT

							14:// LREAL

							20://LWORD

							23://LINT

							11://Date Time-- Needs casting.
								//B&R Casting Returns #DTxx xx xx xx
								//We need to return the C# Standard DT format,, Date..T...Time
								brsmemcpy(ADR(val),pv_Adr,pv_dataLen);
								tempString := DATE_TO_STRING(DT_TO_DATE(UDINT_TO_DT(val)));
								pv_dataLen := brsstrlen(ADR(tempString));
								elementVal := RIGHT(tempString,UDINT_TO_INT(pv_dataLen - 2));

								brsstrcat(ADR(elementVal),ADR('T'));

								tempString := TOD_TO_STRING(DT_TO_TOD(UDINT_TO_DT(val)));
								pv_dataLen := brsstrlen(ADR(tempString));
								tempString := RIGHT(tempString,UDINT_TO_INT(pv_dataLen - 4));
								brsstrcat(ADR(elementVal),ADR(tempString));

							12://Time Only
								elementVal := 'Time';
							13://Date only
								elementVal := 'Date';
							16://Time of day
								elementVal := 'Time Of Day';
							15://Array of structure- We could have to decode futher into here
								//For now we just write this with no data.
								state := READ_DATA_STRUCTURE;
								index := index + 1;

						END_CASE;
					ELSIF pvGetAdrStatus <> ERR_FUB_BUSY THEN
						state := CLOSE_WRITER;
						LastError := pvGetAdrStatus;
					END_IF;
				ELSIF (pvStatus <> ERR_FUB_BUSY) THEN
					state := CLOSE_WRITER;
					LastError := pvStatus;
				END_IF;
			ELSIF xmlWriteElementStart.status <> ERR_FUB_BUSY THEN
				state := CLOSE_WRITER;
				LastError := xmlWriteElementStart.status;
			END_IF;

		WRITE_ELEMENT_TEXT:
			//Write the PV value into the elements..
			xmlWriteElemText.enable := 1;
			xmlWriteElemText.ident := ident;
			xmlWriteElemText.pText := ADR(elementVal);
			xmlWriteElemText();
			IF (xmlWriteElemText.status = ERR_OK) THEN
				state := WRITE_END_ELEMENT;
			ELSIF (xmlWriteElemText.status <> ERR_FUB_BUSY) THEN
				state := CLOSE_WRITER;
				LastError := xmlWriteElemText.status;
			END_IF;

		WRITE_END_ELEMENT: //Only close element with a value..
			xmlWriteEndElement.enable := 1;
			xmlWriteEndElement.ident := ident;
			xmlWriteEndElement();
			IF (xmlWriteEndElement.status = ERR_OK) THEN
				openElements := openElements - 1;
				state := READ_DATA_STRUCTURE;
				index := index + 1;// Get the next piece of data.
			ELSIF (xmlWriteEndElement.status <> ERR_FUB_BUSY) THEN
				LastError := xmlWriteEndElement.status;
				state := CLOSE_WRITER;
			END_IF;

		CLOSE_ALL_ELEMENTS://Close all remaining open elements.
			IF (openElements >= 1) THEN
				xmlWriteEndElement.enable := 1;
				xmlWriteEndElement.ident := ident;
				xmlWriteEndElement();
				IF (xmlWriteEndElement.status = ERR_OK) THEN
					openElements := openElements - 1;
				ELSIF (xmlWriteEndElement.status <> ERR_FUB_BUSY) THEN
					LastError := xmlWriteEndElement.status;
					state := CLOSE_WRITER;
				END_IF;
			ELSE
				state := END_DOC;
			END_IF;

		END_DOC://
			xmlEndDocument.enable := 1;
			xmlEndDocument.ident := ident;
			xmlEndDocument();
			IF (xmlEndDocument.status = ERR_OK) THEN
				state := CREATE_XML_FILE;
			ELSIF (xmlEndDocument.status <> ERR_FUB_BUSY) THEN
				LastError := xmlEndDocument.status;
				state := CLOSE_WRITER;
			END_IF;

		CREATE_XML_FILE://Copy the XML file to the required data area.
			xmlGetMemInfo.enable := 1;
			xmlGetMemInfo.ident := ident;
			xmlGetMemInfo();
			IF (xmlGetMemInfo.status = ERR_OK) THEN
				IF (sizeData >= xmlGetMemInfo.xmlDataSize) THEN
					//memcpy(pData,xmlGetMemInfo.pXmlData,xmlGetMemInfo.xmlDataSize);
					brsstrcpy(pData,xmlGetMemInfo.pXmlData);
					state := CLOSE_WRITER;
				ELSE
					LastError := 1001;//Data area to small.
					state := CLOSE_WRITER;
				END_IF;
			ELSIF (xmlGetMemInfo.status <> ERR_FUB_BUSY) THEN
				LastError := xmlGetMemInfo.status;
				state := CLOSE_WRITER;
			END_IF;

		CLOSE_WRITER://
			xmlCloseWriter.enable := 1;
			xmlCloseWriter.ident := ident;
			IF (xmlCloseWriter.status = ERR_OK) THEN
				ident := 0;
				IF LastError = 0 THEN
					state := FINISHED;
				ELSE
					state := ERROR;
				END_IF;
			ELSIF (xmlCloseWriter.status <> ERR_FUB_BUSY) THEN
				ident := 0;
				state := ERROR;
			END_IF;

		FINISHED:
			status := ERR_OK;

		ERROR:
			status := LastError;

	END_CASE;
	IF (LastError > 0) THEN
		status := LastError;
	END_IF;

END_FUNCTION_BLOCK
```

### Variables.var
```iecst
VAR CONSTANT
	ERR_SYS_PV_NOT_FOUND : UINT := 14710;
END_VAR
```

### Program Logical/File_System/zzFileTransfer (IEC)

#### Variables.var
```iecst
VAR
	state : UINT;
	adrFileName : UDINT;
END_VAR
VAR CONSTANT
	MEMCARD_SAVE : UINT := 1;
	MEMCARD_READ : UINT := 2;
END_VAR
VAR
	adrFileDevice : UDINT;
	init : UINT;
	devLink : DevLink;
	adrParameter : UDINT;
	fileRW : fileReadWrite;
	TestData : ARRAY[0..99] OF USINT;
	do_GetInfo : DatObjInfo;
	error : UINT;
	do_Read : DatObjRead;
	testSize : UDINT;
	do_Create : DatObjCreate;
	do_Delete : DatObjDelete;
	do_Ident : UDINT;
	fiToDatObj : fileToDatObj;
	do_Write : DatObjWrite;
	xmlReadCreate : xmlCreateMemoryReader;
	xmlReadNode : xmlReadNextNode;
	forceRead : BOOL;
	skip : BOOL;
	xmlName : STRING[100];
	xmlValue : STRING[100];
	xmlReadAttNum : xmlReadAttributeNr;
	xmlIndex : UDINT;
	xmlCloseReader : xmlCloseMemoryReader;
	fiToMem : fileToMem;
	pTempMem : UDINT;
	sizeTempMem : UDINT;
	xmlReader : UINT;
	xmlProperty : STRING[100];
	xmlPropertyIndex : DINT;
	n : UINT;
	lineCount : UDINT;
END_VAR
```

#### Main.st
```iecst
(********************************************************************
 * COPYRIGHT --
 ********************************************************************
 * PROGRAM: pnlMemCard
 * File: pnlMemCard.st
 * Author: treamsbottom
 * Created: April 8, 2016
 ********************************************************************
 * Implementation OF PROGRAM pnlMemCard
 ********************************************************************)

PROGRAM _INIT
	state 			:= 0;
	adrFileName 	:= ADR('Test');//file name
	adrFileDevice	:= ADR('memcard');  //ADR('FTP');//Can be file name set up in AS, or Devlink folder name
	//adrParameter := ADR('/DEVICE=C:\\Projects\FTP\Test');//Path for Devlink
	//adrParameter := ADR('/SIP=10.8.4.211 /PROTOCOL=ftp /USER=SUP /PASSWORD=12345');
	//Create temporary memory object for the files to be read into..
	sizeTempMem := 30000000; //Allocate 30MB of free memory
	TMP_alloc(sizeTempMem,ADR(pTempMem));
	init := 1;
END_PROGRAM

PROGRAM _CYCLIC
	IF init = 1 THEN
		//Get pointer to device. not using AS
//		devLink.enable := 1;
//		devLink.pDevice := adrFileDevice;
//		devLink.pParam := adrParameter;
//		devLink();
//		IF (devLink.status = ERR_OK) OR (devLink.status = fiERR_DEVICE_ALREADY_EXIST) THEN
			init:= 0;
//		ELSIF devLink.status = fiERR_SYSTEM THEN
//			error := FileIoGetSysError();
//		END_IF;
	ELSE
		CASE state OF
			MEMCARD_SAVE:
				fileRW.enable := 1;
				fileRW.mode := FILE_SAVE;
				fileRW.pFileDevice := adrFileDevice;
				fileRW.pFileName := ADR('line') ;//adrFileName;
				fileRW.pData := ADR(Line[0]);
				fileRW.sizeData := SIZEOF(Line);
				fileRW.Offset := 0;
				fileRW();
				IF fileRW.status = ERR_OK THEN
					state := 99;
				ELSIF fileRW.status <> ERR_FUB_BUSY THEN
					state := 100;
				END_IF;

			MEMCARD_READ:
				fileRW.enable := 1;
				fileRW.mode := FILE_READ;
				fileRW.pFileDevice := adrFileDevice;
				fileRW.pFileName := adrFileName;
				fileRW.pData := do_Ident;//ADR(TestData[0]);
				fileRW.sizeData := testSize;//SIZEOF(TestData);//100;
				fileRW.Offset := 0;
				fileRW();
				IF fileRW.status = ERR_OK THEN
					state := 99;
				ELSIF fileRW.status <> ERR_FUB_BUSY THEN
					state := 100;
				END_IF;

//			5:
//				do_Read.enable := 1;
//				do_Read.ident := do_Ident;
//				do_Read.pDestination := ADR(TestData[0]);
//				do_Read.len := 99;//testSize;
//				do_Read();
//				IF do_Read.status = ERR_OK	THEN
//					state := 99;
//				ELSIF do_Read.status <> ERR_FUB_BUSY THEN
//					state := 100;
//				END_IF;
//
//			6:
//				//Test get address of data object ot see if we can copy the data we need into data object
//				do_GetInfo.enable := 1;
//				do_GetInfo.pName := ADR('Config');
//				do_GetInfo();
//				IF do_GetInfo.status = ERR_OK THEN
//					do_Ident := do_GetInfo.ident;
//					state := 99;
//				ELSIF do_GetInfo.status <> ERR_FUB_BUSY THEN
//					state := 100;
//				END_IF;
//
//
//			7:
//				do_Create.enable 	:= 1;
//				do_Create.pName 	:= ADR('Config');
//				do_Create.Option 	:= doNO_CS;// DO NOT USE CHECKSUM AS WE COPY DATA DIRECTLY IN THE MEMORY..
//				do_Create.pCpyData 	:= 0;
//				do_Create.MemType	:= doUSRROM;
//				do_Create.len		:= testSize;
//				do_Create();
//				IF (do_Create.status = ERR_OK) OR (do_Create.status = doERR_CHECKSUM_WARNING) THEN
//					do_Ident := do_Create.ident;
//					state := 99;
//				ELSIF do_Create.status <> ERR_FUB_BUSY THEN
//					state := 100;
//				END_IF;
//
//			8:
//				do_Delete.enable := 1;
//				do_Delete.ident := do_Ident;
//				do_Delete();
//				IF do_Delete.status = ERR_OK THEN
//					state := 99;
//				ELSIF do_Delete.status <> ERR_FUB_BUSY THEN
//					state := 100;
//				END_IF;

			10:
//				fiToDatObj.enable := 1;
//				fiToDatObj.pFileDevice := adrFileDevice;
//				fiToDatObj.pFileName := ADR('Test');// adrFileName;
//				fiToDatObj.pDoName := ADR('Config');
//				fiToDatObj.MemType := doUSRROM;
//				fiToDatObj();
//				IF fiToDatObj.status = ERR_OK THEN
//					state := 99;
//				ELSIF fiToDatObj.status <> ERR_FUB_BUSY THEN
//					state := 100;
//				END_IF;
				fiToMem.enable := 1;
				fiToMem.pFileDevice := adrFileDevice;
				fiToMem.pFileName := adrFileName;
				fiToMem.pTempMem := pTempMem;
				fiToMem.sizeTempMem := sizeTempMem;
				fiToMem();
				IF fiToMem.status = ERR_OK THEN
					state := 99;
				ELSIF fiToMem.status <> ERR_FUB_BUSY THEN
					state := 100;
				END_IF;

			11:
//				do_Write.enable := 1;
//				do_Write.ident := do_Ident;
//				do_Write.Offset := 0;
//				do_Write.len := do_GetInfo.len;
//				do_Write.pSource := do_GetInfo.pDatObjMem;
//				do_Write();
//				IF do_Write.status = ERR_OK	 THEN
//					state := 99;
//				ELSIF do_Write.status <> ERR_FUB_BUSY THEN
//					state := 100;
//				END_IF;

			12: //Create XML Readt
				xmlReadCreate.enable := 1;
				xmlReadCreate.memorySize := fiToMem.fiSize;
				xmlReadCreate.pXmlMemory := pTempMem;
				xmlReadCreate();
				IF xmlReadCreate.status = ERR_OK THEN
					state := 99;
				ELSIF xmlReadCreate.status <> ERR_FUB_BUSY THEN
					state := 100;
				END_IF;

			13:	//Read next node
				xmlReadNode.enable := 1;
				xmlReadNode.ident := xmlReadCreate.ident;
				xmlReadNode.forceRead := forceRead;
				xmlReadNode.skipSubtree := skip;
				xmlReadNode.pName := ADR(xmlName);
				xmlReadNode.nameSize := SIZEOF(xmlName);
				xmlReadNode.pValue := ADR(xmlValue);
				xmlReadNode.valueSize := SIZEOF(xmlValue);
				xmlReadNode();
				IF xmlReadNode.status = ERR_OK THEN
					state := 99;
				ELSIF xmlReadNode.status <> ERR_FUB_BUSY THEN
					state := 100;
				END_IF

			14://Read Attribute number
				xmlReadAttNum.enable := 1;
				xmlReadAttNum.ident := xmlReadCreate.ident;
				xmlReadAttNum.index := xmlIndex;
				xmlReadAttNum.pName := ADR(xmlName);
				xmlReadAttNum.nameSize := SIZEOF(xmlName);
				xmlReadAttNum.pValue := ADR(xmlValue);
				xmlReadAttNum.valueSize := SIZEOF(xmlValue);
				xmlReadAttNum();
				IF xmlReadAttNum.status = ERR_OK THEN
					state := 99;
				ELSIF xmlReadAttNum.status <> ERR_FUB_BUSY THEN
					state := 100;
				END_IF

			15:
				xmlCloseReader.enable := 1;
				xmlCloseReader.ident := xmlReadCreate.ident;
				xmlCloseReader();
				IF xmlCloseReader.status = ERR_OK THEN
					state := 99;
				ELSIF xmlCloseReader.status <> ERR_FUB_BUSY THEN
					state := 100;
				END_IF;

			20:
			n:= 0;
			FOR n:= 0 TO 100 DO //Use loop to increase scan time..
				CASE xmlReader OF
					0://Copy into memory
						fiToMem.enable := 1;
						fiToMem.pFileDevice := adrFileDevice;
						fiToMem.pFileName := adrFileName;
						fiToMem.pTempMem := pTempMem;
						fiToMem.sizeTempMem := sizeTempMem;
						fiToMem();
						IF fiToMem.status = ERR_OK THEN
							xmlReader := 1;
						ELSIF fiToMem.status <> ERR_FUB_BUSY THEN
							xmlReader := 100;
						END_IF;

					1://Create XML Reaser
						xmlReadCreate.enable := 1;
						xmlReadCreate.memorySize := fiToMem.fiSize;
						xmlReadCreate.pXmlMemory := pTempMem;
						xmlReadCreate();
						IF xmlReadCreate.status = ERR_OK THEN
							lineCount := 0;
							xmlReader := 2;
						ELSIF xmlReadCreate.status <> ERR_FUB_BUSY THEN
							xmlReader := 100;
						END_IF;

					2://Search for 'Config setting'
						xmlReadNode.enable := 1;
						xmlReadNode.ident := xmlReadCreate.ident;
						xmlReadNode.forceRead := forceRead;
						xmlReadNode.skipSubtree := skip;
						xmlReadNode.pName := ADR(xmlName);
						xmlReadNode.nameSize := SIZEOF(xmlName);
						xmlReadNode.pValue := ADR(xmlValue);
						xmlReadNode.valueSize := SIZEOF(xmlValue);
						xmlReadNode();
						IF xmlReadNode.status = ERR_OK THEN
							IF xmlName = 'Config' THEN
								lineCount := lineCount + 1;
								xmlIndex := 0;
								xmlReader := 3;
							END_IF;
						ELSIF xmlReadNode.status = xmlERR_NO_FURTHER_XML_NODE THEN
							xmlReader := 4;//End of file
						ELSIF xmlReadNode.status <> ERR_FUB_BUSY THEN
							xmlReader := 100;
						END_IF

					3://Decode XML elements
						xmlReadAttNum.enable := 1;
						xmlReadAttNum.ident := xmlReadCreate.ident;
						xmlReadAttNum.index := xmlIndex;
						xmlReadAttNum.pName := ADR(xmlName);
						xmlReadAttNum.nameSize := SIZEOF(xmlName);
						xmlReadAttNum.pValue := ADR(xmlValue);
						xmlReadAttNum.valueSize := SIZEOF(xmlValue);
						xmlReadAttNum();
						IF xmlReadAttNum.status = ERR_OK THEN
							IF xmlName = 'Property' THEN
									xmlProperty := xmlValue;
							ELSIF xmlName = 'Index' THEN
								xmlPropertyIndex := atoi(ADR(xmlValue));
							ELSIF xmlName =	'FirstBag' THEN
								IF (xmlProperty = 'Line') AND (xmlPropertyIndex > 0) AND  (xmlPropertyIndex <= MAX_LINES) THEN
									Line[xmlPropertyIndex].FirstBag := DINT_TO_UINT(atoi(ADR(xmlValue)));
								END_IF;
							ELSIF xmlName = 'LastBag' THEN
								IF (xmlProperty = 'Line') AND (xmlPropertyIndex > 0) AND  (xmlPropertyIndex <= MAX_LINES) THEN
									Line[xmlPropertyIndex].LastBag := DINT_TO_UINT(atoi(ADR(xmlValue)));
								END_IF;
							END_IF;
							xmlIndex := xmlIndex + 1;
						ELSIF xmlReadAttNum.status = xmlERR_INVALID_ATTRIBUTE_INDEX THEN//No more elements go back to beginning..
							xmlReader := 2;
						ELSIF xmlReadAttNum.status <> ERR_FUB_BUSY THEN
							xmlReader := 100;
						END_IF

					4://Close XML Reader
						xmlCloseReader.enable := 1;
						xmlCloseReader.ident := xmlReadCreate.ident;
						xmlCloseReader();
						IF xmlCloseReader.status = ERR_OK THEN
							xmlReader := 99;
						ELSIF xmlCloseReader.status <> ERR_FUB_BUSY THEN
							xmlReader := 100;
						END_IF;

					99:
						state := 99;
						xmlReader := 0;
					100://Error
						state := 100;
						xmlReader := 0;

				END_CASE;
				IF xmlReader = 0 THEN
					EXIT;
				END_IF;
			END_FOR;

		END_CASE;
	END_IF;

END_PROGRAM
```

### Program Logical/File_System/zzXMLFile (IEC)

#### Variables.var
```iecst
(*State Constants*)
VAR CONSTANT
	XML_READER_IDLE : UINT := 0;
	XML_READER_COPY_FILE_TO_MEMCARD : UINT := 1;
	XML_READER_DECODE_FILE : UINT := 2;
	XML_READER_DECODE_ERROR : UINT := 99;
END_VAR
(**Local Vars*)
VAR
	state : UINT;
	error : UINT;
	pTempMem : UDINT;
	sizeTempMem : UDINT;
	pFileName : UDINT;
	pFileDevice : UDINT;
	pDevLinkParameter : UDINT;
	pMemCard : UDINT;
	fileCopyFromDev : FileCopyFromDev;
	pUSB : UDINT;
	n : UINT;
	xmlReader : UINT;
	lineCount : UINT;
	xmlName : STRING[100];
	xmlValue : STRING[100];
	xmlIndex : UDINT;
	xmlProperty : STRING[100];
	xmlPropertyIndex : DINT;
	fiToMem : fileToMem;
	xmlReadCreate : xmlCreateMemoryReader;
	xmlReadNode : xmlReadNextNode;
	xmlReadAttNum : xmlReadAttributeNr;
	xmlCloseReader : xmlCloseMemoryReader;
	testString : STRING[100];
	fileWrite : fileReadWrite;
END_VAR
```
